METHOD dataProcessing : BOOL
VAR_INPUT
END_VAR
VAR
	i_CGResult:INT;
	i_HResult:INT;
	str1:STRING;
END_VAR
FOR logHandleArray_index:=1 TO logHandleArrayLength DO
	CASE nSocketType OF
	0://TCPIP server
		str1:=CONCAT(str1,BYTE_TO_HEXSTR(tcpipRecData.b1,2,FALSE));
		str1:=CONCAT(str1,' ');
		str1:=CONCAT(str1,BYTE_TO_HEXSTR(tcpipRecData.b2,2,FALSE));
		str1:=CONCAT(str1,' ');
		str1:=CONCAT(str1,BYTE_TO_HEXSTR(tcpipRecData.b3,2,FALSE));
		str1:=CONCAT(str1,' ');
		str1:=CONCAT(str1,BYTE_TO_HEXSTR(tcpipRecData.b4,2,FALSE));
		str1:=CONCAT(str1,' ');
		str1:=CONCAT(str1,BYTE_TO_HEXSTR(tcpipRecData.b5,2,FALSE));
		str1:=CONCAT(str1,' ');
		str1:=CONCAT(str1,BYTE_TO_HEXSTR(tcpipRecData.b6,2,FALSE));
		str1:=CONCAT(str1,' ');
		str1:=CONCAT(str1,BYTE_TO_HEXSTR(tcpipRecData.b7,2,FALSE));
		str1:=CONCAT(str1,' ');
		str1:=CONCAT(str1,BYTE_TO_HEXSTR(tcpipRecData.b8,2,FALSE));
		str1:=CONCAT(str1,' ');
		str1:=CONCAT(str1,BYTE_TO_HEXSTR(tcpipRecData.b9,2,FALSE));
		str1:=CONCAT(str1,' ');
		str1:=CONCAT(str1,BYTE_TO_HEXSTR(tcpipRecData.b10,2,FALSE));
		str1:=CONCAT(str1,' ');
		str1:=CONCAT(str1,BYTE_TO_HEXSTR(tcpipRecData.b11,2,FALSE));
		str1:=CONCAT(str1,' ');
		str1:=CONCAT(str1,BYTE_TO_HEXSTR(tcpipRecData.b12,2,FALSE));
		str1:=CONCAT(str1,' ');
		str1:=CONCAT(str1,BYTE_TO_HEXSTR(tcpipRecData.b13,2,FALSE));
		str1:=CONCAT(str1,' ');
		str1:=CONCAT(str1,BYTE_TO_HEXSTR(tcpipRecData.b14,2,FALSE));
		str1:=CONCAT(str1,' ');
		str1:=CONCAT(str1,BYTE_TO_HEXSTR(tcpipRecData.b15,2,FALSE));
		str1:=CONCAT(str1,' ');
		str1:=CONCAT(str1,BYTE_TO_HEXSTR(tcpipRecData.b16,2,FALSE));
		str1:=CONCAT(str1,' ');
		str1:=CONCAT(str1,BYTE_TO_HEXSTR(tcpipRecData.b17,2,FALSE));
		str1:=CONCAT(str1,' ');
		str1:=CONCAT(str1,BYTE_TO_HEXSTR(tcpipRecData.b18,2,FALSE));
		str1:=CONCAT(str1,' ');
		str1:=CONCAT(str1,BYTE_TO_HEXSTR(tcpipRecData.b19,2,FALSE));
		str1:=CONCAT(str1,' ');
		str1:=CONCAT(str1,BYTE_TO_HEXSTR(tcpipRecData.b20,2,FALSE));
//		logHandleArray[logHandleArray_index]^.append(CONCAT(CONCAT(CONCAT('Recevie From ', sTerminalName), ' -- '),str1));
	1://TCPIP client
		str1:=CONCAT(str1,BYTE_TO_HEXSTR(tcpipRecData.b1,2,FALSE));
		str1:=CONCAT(str1,' ');
		str1:=CONCAT(str1,BYTE_TO_HEXSTR(tcpipRecData.b2,2,FALSE));
		str1:=CONCAT(str1,' ');
		str1:=CONCAT(str1,BYTE_TO_HEXSTR(tcpipRecData.b3,2,FALSE));
		str1:=CONCAT(str1,' ');
		str1:=CONCAT(str1,BYTE_TO_HEXSTR(tcpipRecData.b4,2,FALSE));
		str1:=CONCAT(str1,' ');
		str1:=CONCAT(str1,BYTE_TO_HEXSTR(tcpipRecData.b5,2,FALSE));
		str1:=CONCAT(str1,' ');
		str1:=CONCAT(str1,BYTE_TO_HEXSTR(tcpipRecData.b6,2,FALSE));
		str1:=CONCAT(str1,' ');
		str1:=CONCAT(str1,BYTE_TO_HEXSTR(tcpipRecData.b7,2,FALSE));
		str1:=CONCAT(str1,' ');
		str1:=CONCAT(str1,BYTE_TO_HEXSTR(tcpipRecData.b8,2,FALSE));
		str1:=CONCAT(str1,' ');
		str1:=CONCAT(str1,BYTE_TO_HEXSTR(tcpipRecData.b9,2,FALSE));
		str1:=CONCAT(str1,' ');
		str1:=CONCAT(str1,BYTE_TO_HEXSTR(tcpipRecData.b10,2,FALSE));
		str1:=CONCAT(str1,' ');
		str1:=CONCAT(str1,BYTE_TO_HEXSTR(tcpipRecData.b11,2,FALSE));
		str1:=CONCAT(str1,' ');
		str1:=CONCAT(str1,BYTE_TO_HEXSTR(tcpipRecData.b12,2,FALSE));
		str1:=CONCAT(str1,' ');
		str1:=CONCAT(str1,BYTE_TO_HEXSTR(tcpipRecData.b13,2,FALSE));
		str1:=CONCAT(str1,' ');
		str1:=CONCAT(str1,BYTE_TO_HEXSTR(tcpipRecData.b14,2,FALSE));
		str1:=CONCAT(str1,' ');
		str1:=CONCAT(str1,BYTE_TO_HEXSTR(tcpipRecData.b15,2,FALSE));
		str1:=CONCAT(str1,' ');
		str1:=CONCAT(str1,BYTE_TO_HEXSTR(tcpipRecData.b16,2,FALSE));
		str1:=CONCAT(str1,' ');
		str1:=CONCAT(str1,BYTE_TO_HEXSTR(tcpipRecData.b17,2,FALSE));
		str1:=CONCAT(str1,' ');
		str1:=CONCAT(str1,BYTE_TO_HEXSTR(tcpipRecData.b18,2,FALSE));
		str1:=CONCAT(str1,' ');
		str1:=CONCAT(str1,BYTE_TO_HEXSTR(tcpipRecData.b19,2,FALSE));
		str1:=CONCAT(str1,' ');
		str1:=CONCAT(str1,BYTE_TO_HEXSTR(tcpipRecData.b20,2,FALSE));
//		logHandleArray[logHandleArray_index]^.append(CONCAT(CONCAT(CONCAT('Recevie From ', sTerminalName), ' -- '),str1));
	END_CASE
END_FOR

// 数据处理
readStateFlag:=TRUE;
volt:=TO_REAL((tcpipRecData.b10*256+tcpipRecData.b11)/4096.0)*10.0;
dworld:=tcpipRecData.b10*256+tcpipRecData.b11;
END_METHOD

ACTION Manual:
(*
rTrig_Version(CLK:=bTrig_Version);
IF rTrig_Version.Q THEN
	appendSend(0,0,E_CmdID_SW.SW_GetVer,0.0,0.0,0.0,0.0,0.0,0,'');
END_IF
*)
END_ACTION

METHOD PRIVATE popup : BOOL
VAR_INPUT
END_VAR
CASE popupStep OF
0:
	IF (sendPoint<endPoint OR passMax) AND bSendCondition THEN
		popupSendData:=sendDataArray[sendPoint];
		sendData(popupSendData);//此处是调用信息发送
		popupStep:=10;
		sendPoint:=sendPoint+1;
		IF sendPoint>(cNumEnd-1) THEN
			sendPoint:=1;
			passMax:=FALSE;
		END_IF
	END_IF
10:
	popupTON2(IN:=NOT popupTON2.Q, PT:=T#2S);
	IF NOT bSendCondition OR popupTON2.Q THEN
		popupTON2(IN:=FALSE);
		popupStep:=11;
	END_IF
11:
	IF bSendCondition THEN
		popupStep:=12;
	END_IF
	popupTON1(IN:=FALSE);
12:
	//popupTON1(IN:=NOT popupTON1.Q,PT:=T#10MS);
	popupTON1(IN:=NOT popupTON1.Q,PT:=TO_TIME(nQueueInterval));
	IF popupTON1.Q THEN
		popupStep:=0;
	END_IF
END_CASE
END_METHOD

METHOD ReadVoltage : BOOL
VAR_INPUT
END_VAR
appendSend(16#00,16#00,16#00,16#00,16#00,16#06,16#01,16#04,16#00,16#00,16#00,16#04,0,0,0,0,0,0,0,0,12);// 读进电压字符串
END_METHOD

METHOD PRIVATE sendData : BOOL
VAR_INPUT
	dataStruct	:struct_byte;
END_VAR
VAR
	str1:STRING;
END_VAR
IF bSendCondition AND bEnable THEN
	tcpipSendData.b1	:=dataStruct.b1;
	tcpipSendData.b2	:=dataStruct.b2;
	tcpipSendData.b3	:=dataStruct.b3;
	tcpipSendData.b4	:=dataStruct.b4;
	tcpipSendData.b5	:=dataStruct.b5;
	tcpipSendData.b6	:=dataStruct.b6;
	tcpipSendData.b7	:=dataStruct.b7;
	tcpipSendData.b8	:=dataStruct.b8;
	tcpipSendData.b9	:=dataStruct.b9;
	tcpipSendData.b10	:=dataStruct.b10;
	tcpipSendData.b11	:=dataStruct.b11;
	tcpipSendData.b12	:=dataStruct.b12;
	tcpipSendData.b13	:=dataStruct.b13;
	tcpipSendData.b14	:=dataStruct.b14;
	tcpipSendData.b15	:=dataStruct.b15;
	tcpipSendData.b16	:=dataStruct.b16;
	tcpipSendData.b17	:=dataStruct.b17;
	tcpipSendData.b18	:=dataStruct.b18;
	tcpipSendData.b19	:=dataStruct.b19;
	tcpipSendData.b20	:=dataStruct.b20;
	
	CASE nSocketType OF
	0://TCPIP server
		tcpipSendDataBuff_Server:=tcpipSendData;
		tcpipSendData:=tcpipSendDataClear;	
		tcpipServer.bSend:=TRUE;
	1://TCPIP client
		tcpipSendDataBuff_Client:=tcpipSendData;
		tcpipSendData:=tcpipSendDataClear;	
		tcpipClient.bSend:=TRUE;
	END_CASE
	
	FOR logHandleArray_index:=1 TO logHandleArrayLength DO
		CASE nSocketType OF
		0://TCPIP server
			str1:=CONCAT(str1,BYTE_TO_HEXSTR(tcpipSendDataBuff_Server.b1,2,FALSE));
			str1:=CONCAT(str1,' ');
			str1:=CONCAT(str1,BYTE_TO_HEXSTR(tcpipSendDataBuff_Server.b2,2,FALSE));
			str1:=CONCAT(str1,' ');
			str1:=CONCAT(str1,BYTE_TO_HEXSTR(tcpipSendDataBuff_Server.b3,2,FALSE));
			str1:=CONCAT(str1,' ');
			str1:=CONCAT(str1,BYTE_TO_HEXSTR(tcpipSendDataBuff_Server.b4,2,FALSE));
			str1:=CONCAT(str1,' ');
			str1:=CONCAT(str1,BYTE_TO_HEXSTR(tcpipSendDataBuff_Server.b5,2,FALSE));
			str1:=CONCAT(str1,' ');
			str1:=CONCAT(str1,BYTE_TO_HEXSTR(tcpipSendDataBuff_Server.b6,2,FALSE));
			str1:=CONCAT(str1,' ');
			str1:=CONCAT(str1,BYTE_TO_HEXSTR(tcpipSendDataBuff_Server.b7,2,FALSE));
			str1:=CONCAT(str1,' ');
			str1:=CONCAT(str1,BYTE_TO_HEXSTR(tcpipSendDataBuff_Server.b8,2,FALSE));
			str1:=CONCAT(str1,' ');
			str1:=CONCAT(str1,BYTE_TO_HEXSTR(tcpipSendDataBuff_Server.b9,2,FALSE));
			str1:=CONCAT(str1,' ');
			str1:=CONCAT(str1,BYTE_TO_HEXSTR(tcpipSendDataBuff_Server.b10,2,FALSE));
			str1:=CONCAT(str1,' ');
			str1:=CONCAT(str1,BYTE_TO_HEXSTR(tcpipSendDataBuff_Server.b11,2,FALSE));
			str1:=CONCAT(str1,' ');
			str1:=CONCAT(str1,BYTE_TO_HEXSTR(tcpipSendDataBuff_Server.b12,2,FALSE));
			str1:=CONCAT(str1,' ');
			str1:=CONCAT(str1,BYTE_TO_HEXSTR(tcpipSendDataBuff_Server.b13,2,FALSE));
			str1:=CONCAT(str1,' ');
			str1:=CONCAT(str1,BYTE_TO_HEXSTR(tcpipSendDataBuff_Server.b14,2,FALSE));
			str1:=CONCAT(str1,' ');
			str1:=CONCAT(str1,BYTE_TO_HEXSTR(tcpipSendDataBuff_Server.b15,2,FALSE));
			str1:=CONCAT(str1,' ');
			str1:=CONCAT(str1,BYTE_TO_HEXSTR(tcpipSendDataBuff_Server.b16,2,FALSE));
			str1:=CONCAT(str1,' ');
			str1:=CONCAT(str1,BYTE_TO_HEXSTR(tcpipSendDataBuff_Server.b17,2,FALSE));
			str1:=CONCAT(str1,' ');
			str1:=CONCAT(str1,BYTE_TO_HEXSTR(tcpipSendDataBuff_Server.b18,2,FALSE));
			str1:=CONCAT(str1,' ');
			str1:=CONCAT(str1,BYTE_TO_HEXSTR(tcpipSendDataBuff_Server.b19,2,FALSE));
			str1:=CONCAT(str1,' ');
			str1:=CONCAT(str1,BYTE_TO_HEXSTR(tcpipSendDataBuff_Server.b20,2,FALSE));
//			logHandleArray[logHandleArray_index]^.append(CONCAT(CONCAT(CONCAT('Send To ', sTerminalName), ' -- '),str1));
		1://TCPIP client
			str1:=CONCAT(str1,' ');
			str1:=CONCAT(str1,BYTE_TO_HEXSTR(tcpipSendDataBuff_Client.b1,2,FALSE));
			str1:=CONCAT(str1,' ');
			str1:=CONCAT(str1,BYTE_TO_HEXSTR(tcpipSendDataBuff_Client.b2,2,FALSE));
			str1:=CONCAT(str1,' ');
			str1:=CONCAT(str1,BYTE_TO_HEXSTR(tcpipSendDataBuff_Client.b3,2,FALSE));
			str1:=CONCAT(str1,' ');
			str1:=CONCAT(str1,BYTE_TO_HEXSTR(tcpipSendDataBuff_Client.b4,2,FALSE));
			str1:=CONCAT(str1,' ');
			str1:=CONCAT(str1,BYTE_TO_HEXSTR(tcpipSendDataBuff_Client.b5,2,FALSE));
			str1:=CONCAT(str1,' ');
			str1:=CONCAT(str1,BYTE_TO_HEXSTR(tcpipSendDataBuff_Client.b6,2,FALSE));
			str1:=CONCAT(str1,' ');
			str1:=CONCAT(str1,BYTE_TO_HEXSTR(tcpipSendDataBuff_Client.b7,2,FALSE));
			str1:=CONCAT(str1,' ');
			str1:=CONCAT(str1,BYTE_TO_HEXSTR(tcpipSendDataBuff_Client.b8,2,FALSE));
			str1:=CONCAT(str1,' ');
			str1:=CONCAT(str1,BYTE_TO_HEXSTR(tcpipSendDataBuff_Client.b9,2,FALSE));
			str1:=CONCAT(str1,' ');
			str1:=CONCAT(str1,BYTE_TO_HEXSTR(tcpipSendDataBuff_Client.b10,2,FALSE));
			str1:=CONCAT(str1,' ');
			str1:=CONCAT(str1,BYTE_TO_HEXSTR(tcpipSendDataBuff_Client.b11,2,FALSE));
			str1:=CONCAT(str1,' ');
			str1:=CONCAT(str1,BYTE_TO_HEXSTR(tcpipSendDataBuff_Client.b12,2,FALSE));
			str1:=CONCAT(str1,' ');
			str1:=CONCAT(str1,BYTE_TO_HEXSTR(tcpipSendDataBuff_Client.b13,2,FALSE));
			str1:=CONCAT(str1,' ');
			str1:=CONCAT(str1,BYTE_TO_HEXSTR(tcpipSendDataBuff_Client.b14,2,FALSE));
			str1:=CONCAT(str1,' ');
			str1:=CONCAT(str1,BYTE_TO_HEXSTR(tcpipSendDataBuff_Client.b15,2,FALSE));
			str1:=CONCAT(str1,' ');
			str1:=CONCAT(str1,BYTE_TO_HEXSTR(tcpipSendDataBuff_Client.b16,2,FALSE));
			str1:=CONCAT(str1,' ');
			str1:=CONCAT(str1,BYTE_TO_HEXSTR(tcpipSendDataBuff_Client.b17,2,FALSE));
			str1:=CONCAT(str1,' ');
			str1:=CONCAT(str1,BYTE_TO_HEXSTR(tcpipSendDataBuff_Client.b18,2,FALSE));
			str1:=CONCAT(str1,' ');
			str1:=CONCAT(str1,BYTE_TO_HEXSTR(tcpipSendDataBuff_Client.b19,2,FALSE));
			str1:=CONCAT(str1,' ');
			str1:=CONCAT(str1,BYTE_TO_HEXSTR(tcpipSendDataBuff_Client.b20,2,FALSE));
//			logHandleArray[logHandleArray_index]^.append(CONCAT(CONCAT(CONCAT('Send To ', sTerminalName), ' -- '),str1));
		END_CASE
	END_FOR
END_IF
END_METHOD

END_PROGRAM

// ---- POUs/Communication/PLC_String.TcPOU
PROGRAM PLC_String
VAR_INPUT
	nSocketType:UINT:=0;// socket 类型; 0 表示 server; 1 表示 client;
	sTerminalName:STRING;// 通讯对方名称 自定义
	sHost:STRING(20):='127.0.0.1';// 通讯IP地址; server时表示本地host; client时表示远程host
	nPort:UDINT:=8900;// 通讯端口号;
	bEnable:BOOL:=TRUE;// 通讯启用\禁用连接
	sSendSuffix:STRING:='';//此处可统一添加发送后缀字符 $R$N
	nQueueInterval:UDINT:=50;// 发送队列时间间隔 单位ms
	logHandleArray:ARRAY [1..5] OF POINTER TO printLogModule_EX;// log 操作 handle 数组
	logHandleArrayLength:UINT:=0;// log 操作 handle 数组长度, 不超过5
END_VAR
VAR_OUTPUT
	bSendCondition	:BOOL;//可发送条件
	bSocketConnected:BOOL;//连接状态
END_VAR
VAR CONSTANT
	cNumBegin		:DINT:=1;
	cNumEnd			:DINT:=100;
END_VAR
VAR
	sendDataArray	:ARRAY [cNumBegin..cNumEnd] OF STRING(255);
	length			:DINT:=0;
	endPoint		:DINT:=cNumBegin;
	popupSendData	:STRING(255);
	//popup
	popupStep		:UINT:=0;
	popupTON1		:TON;
	popupTON2		:TON;
	iPopup			:DINT:=0;
	_PopupLength	:DINT:=0;
END_VAR
VAR
	tcpipClient					:tcpipClientModule_EX;
	tcpipServer					:tcpipServerModule_EX;////定义服务器对象
	
	tcpipSendDataBuff_Server	:STRING(255);//发送数据 Buff server
	tcpipSendDataBuff_Client	:STRING(255);//发送数据 Buff client
	
	tcpipSendDataClear			:STRING(255);//发送数据 清空
	tcpipSendData				:STRING(255);//发送数据
	
	tcpipRecDataBuff_Server		:STRING(255);//已接收数据 Buff server
	tcpipRecDataBuff_Client		:STRING(255);//已接收数据 Buff client
	
	tcpipRecDataClear			:STRING(255);//已接收数据 清空
	tcpipRecData				:STRING(255);//已接收数据
	
	tcpConnectR_Trig			:R_Trig;//初始连接上升沿
	tcpConnectF_Trig			:F_Trig;//初始连接下降沿
	registerStep				:UDINT;//ALC注册控制步
	registerTON					:TON;//ALC注册延时
	
	logHandleArray_index		:UINT:=1;
END_VAR
VAR
	bTrig_Start:BOOL;
	rTrig_Start:R_TRIG;
	tTrig_Start:TON;
	
	bTrig_Stop:BOOL;
	rTrig_Stop:R_TRIG;
	tTrig_Stop:TON;
	
	bTrig_Reset:BOOL;
	rTrig_Reset:R_TRIG;
	tTrig_Reset:TON;
	
	
	bTrig_Init:BOOL;
	rTrig_Init:R_TRIG;
	
	bTrig_All_Home:BOOL;
	rTrig_All_Home:R_TRIG;
	
	bTrig_Z_Safe:BOOL;
	rTrig_Z_Safe:R_TRIG;
	
	bTrig_P_Pos_:BOOL;
	rTrig_P_Pos_:R_TRIG;
	nTrig_P_Pos_TrayNum:UINT:=1;
	nTrig_P_Pos_RowNum:UINT:=1;
	
	bTrig_Move_P_:BOOL;
	rTrig_Move_P_:R_TRIG;
	nTrig_Move_P_TrayNum:UINT:=1;
	nTrig_Move_P_RowNum:UINT:=1;
	nTrig_Move_P_PosNum:UINT:=1;
	findposstart	:INT;
	findposend		:INT;
	find_pos		:INT;
	recStrTemp		:STRING(255);
END_VAR


CASE nSocketType OF
0://TCPIP server
	tcpipServer(
		sSrvNetId:= , 
		sLocalHost:=sHost , 
		nLocalPort:=nPort , 
		bStartConnect:=bEnable , 
		tcpipSDataLen:=TO_UDINT(LEN(tcpipSendDataBuff_Server)) , 
		tcpipSData:=ADR(tcpipSendDataBuff_Server) , 
		bSend:= , 
		tcpipRecDataLen:=SIZEOF(tcpipRecDataBuff_Server) , 
		tcpipRecData:=ADR(tcpipRecDataBuff_Server) , 
		bAccepted=> , 
		bSendBusy=> , 
		bRecData=> );
	bSendCondition:=tcpipServer.bAccepted AND NOT tcpipServer.bSendBusy;
	//TCPIP连接
	bSocketConnected:=tcpipServer.bAccepted;
	IF NOT tcpipServer.bAccepted THEN
		length:=0;
		endPoint:=cNumBegin;
	END_IF
	tcpConnectR_Trig(CLK:=tcpipServer.bAccepted);
	tcpConnectF_Trig(CLK:=tcpipServer.bAccepted);

1://TCPIP client
	tcpipClient(
		sSrvNetId:= , 
		sRemoteHost:=sHost , 
		nRemotePort:=nPort , 
		bStartConnect:=bEnable , 
		tcpipSDataLen:=TO_UDINT(LEN(tcpipSendDataBuff_Client)) , 
		tcpipSData:=ADR(tcpipSendDataBuff_Client) , 
		bSend:= , 
		tcpipRecDataLen:=SIZEOF(tcpipRecDataBuff_Client) , 
		tcpipRecData:=ADR(tcpipRecDataBuff_Client) , 
		bConnected=> , 
		bSendBusy=> , 
		bRecData=> );
	bSendCondition:=tcpipClient.bConnected AND NOT tcpipClient.bSendBusy;
	//TCPIP连接
	bSocketConnected:=tcpipClient.bConnected;
	IF NOT tcpipClient.bConnected THEN
		length:=0;
		endPoint:=cNumBegin;
	END_IF
	tcpConnectR_Trig(CLK:=tcpipClient.bConnected);
	tcpConnectF_Trig(CLK:=tcpipClient.bConnected);
END_CASE

IF tcpConnectR_Trig.Q THEN
	FOR logHandleArray_index:=1 TO logHandleArrayLength DO
		logHandleArray[logHandleArray_index]^.append(CONCAT(sTerminalName, ' has been connected'));
	END_FOR
	registerStep:=10;
END_IF
IF tcpConnectF_Trig.Q THEN
	FOR logHandleArray_index:=1 TO logHandleArrayLength DO
		logHandleArray[logHandleArray_index]^.append(CONCAT(sTerminalName, ' has been disconnected'));
	END_FOR
	registerStep:=0;
END_IF
//数据接收处理
CASE nSocketType OF
0://TCPIP server
	IF tcpipServer.bRecData THEN
		tcpipRecData:=tcpipRecDataBuff_Server;//buff转存
		tcpipRecDataBuff_Server:=tcpipRecDataClear;//转存之后清空buff
		dataProcessing();
	END_IF
1://TCPIP client
	IF tcpipClient.bRecData THEN
		tcpipRecData:=tcpipRecDataBuff_Client;//buff转存
		tcpipRecDataBuff_Client:=tcpipRecDataClear;//转存之后清空buff
		dataProcessing();
	END_IF
END_CASE


popup();

CASE registerStep OF
0:
	//Ready
END_CASE

ACTION ACT_dataProcessing_DOE:
//(*LoadCCD3*)
//	recStrFilArrSocket[1]:='CoaxialCCD1:';
//	recStrFilArrSocket[2]:='DUTTopX:';
//	recStrFilArrSocket[3]:='DUTTopY:';
//	recStrFilArrSocket[4]:='DUTBottomX:';
//	recStrFilArrSocket[5]:='DUTBottomY:';
//	recStrFilArrSocket[6]:='SocketTopX:';
//	recStrFilArrSocket[7]:='SocketTopY:';
//	recStrFilArrSocket[8]:='SocketBottomX:';
//	recStrFilArrSocket[9]:='SocketBottomY:';
//	recStrFilArrSocket[10]:='ModelAngle:';
	
//	recStrTemp:='';
//	find_pos:=FIND(tcpipRecData, recStrFilArrSocket[1]);
//	IF find_pos>0 THEN
//		findposstart:=find_pos;
//		find_pos:=0;
//		find_pos:=FIND(tcpipRecData, ';');
//		IF find_pos>0 THEN
//			findposend:=find_pos;
//			find_pos:=0;
//		END_IF
//		recPosArrSocket_G_CCD1[1]:=STRING_TO_LREAL(MID(tcpipRecData,findposend-findposstart-(len(recStrFilArrSocket[1])+len(recStrFilArrSocket[2])),findposstart+len(recStrFilArrSocket[1])+len(recStrFilArrSocket[2])));
//		recStrTemp:=DELETE(tcpipRecData,findposend-findposstart+1,findposstart);
//		find_pos:=0;
//		findposstart:=1;
//		find_pos:=FIND(recStrTemp, ';');
//		IF find_pos>0 THEN
//			findposend:=find_pos;
//			find_pos:=0;
//		END_IF
//		recPosArrSocket_G_CCD1[2]:=STRING_TO_LREAL(MID(recStrTemp,findposend-findposstart-len(recStrFilArrSocket[3]),findposstart+len(recStrFilArrSocket[3])));
//		recStrTemp:=DELETE(recStrTemp,findposend-findposstart+1,findposstart);
//		find_pos:=0;
//		findposstart:=1;
//		find_pos:=FIND(recStrTemp, ';');
//		IF find_pos>0 THEN
//			findposend:=find_pos;
//			find_pos:=0;
//		END_IF
//		recPosArrSocket_G_CCD1[3]:=STRING_TO_LREAL(MID(recStrTemp,findposend-findposstart-len(recStrFilArrSocket[4]),findposstart+len(recStrFilArrSocket[4])));
//		recStrTemp:=DELETE(recStrTemp,findposend-findposstart+1,findposstart);
//		find_pos:=0;
//		findposstart:=1;
//		find_pos:=FIND(recStrTemp, ';');
//		IF find_pos>0 THEN
//			findposend:=find_pos;
//			find_pos:=0;
//		END_IF
//		recPosArrSocket_G_CCD1[4]:=STRING_TO_LREAL(MID(recStrTemp,findposend-findposstart-len(recStrFilArrSocket[5]),findposstart+len(recStrFilArrSocket[5])));
//		recStrTemp:=DELETE(recStrTemp,findposend-findposstart+1,findposstart);
//		find_pos:=0;
//		findposstart:=1;
//		find_pos:=FIND(recStrTemp, ';');
//		IF find_pos>0 THEN
//			findposend:=find_pos;
//			find_pos:=0;
//		END_IF
//		recPosArrSocket_G_CCD1[5]:=STRING_TO_LREAL(MID(recStrTemp,findposend-findposstart-len(recStrFilArrSocket[6]),findposstart+len(recStrFilArrSocket[6])));
//		recStrTemp:=DELETE(recStrTemp,findposend-findposstart+1,findposstart);
//		find_pos:=0;
//		findposstart:=1;
//		find_pos:=FIND(recStrTemp, ';');
//		IF find_pos>0 THEN
//			findposend:=find_pos;
//			find_pos:=0;
//		END_IF
//		recPosArrSocket_G_CCD1[6]:=STRING_TO_LREAL(MID(recStrTemp,findposend-findposstart-len(recStrFilArrSocket[7]),findposstart+len(recStrFilArrSocket[7])));
//		recStrTemp:=DELETE(recStrTemp,findposend-findposstart+1,findposstart);
//		find_pos:=0;
//		findposstart:=1;
//		find_pos:=FIND(recStrTemp, ';');
//		IF find_pos>0 THEN
//			findposend:=find_pos;
//			find_pos:=0;
//		END_IF
//		recPosArrSocket_G_CCD1[7]:=STRING_TO_LREAL(MID(recStrTemp,findposend-findposstart-len(recStrFilArrSocket[8]),findposstart+len(recStrFilArrSocket[8])));
//		recStrTemp:=DELETE(recStrTemp,findposend-findposstart+1,findposstart);
//		find_pos:=0;
//		findposstart:=1;
//		find_pos:=FIND(recStrTemp, ';');
//		IF find_pos>0 THEN
//			findposend:=find_pos;
//			find_pos:=0;
//		END_IF
//		recPosArrSocket_G_CCD1[8]:=STRING_TO_LREAL(MID(recStrTemp,findposend-findposstart-len(recStrFilArrSocket[9]),findposstart+len(recStrFilArrSocket[9])));
//		recStrTemp:=DELETE(recStrTemp,findposend-findposstart+1,findposstart);
//		find_pos:=0;
//		findposstart:=1;
//		find_pos:=FIND(recStrTemp, ';');
//		IF find_pos>0 THEN
//			findposend:=find_pos;
//			find_pos:=0;
//		END_IF
//		recPosArrSocket_G_CCD1[9]:=STRING_TO_LREAL(MID(recStrTemp,findposend-findposstart-len(recStrFilArrSocket[10]),findposstart+len(recStrFilArrSocket[10])));
//		recStrTemp:=DELETE(recStrTemp,findposend-findposstart+1,findposstart);
//		recCCDResultArr[3]:=TRUE;
//	END_IF
END_ACTION

METHOD appendSend : BOOL
VAR_INPUT
	str			:STRING(255);
END_VAR
VAR
	suffix					:STRING;
	strTemp_appendSend		:STRING(255);
END_VAR

IF endPoint>(cNumEnd-1) THEN
	RETURN;
END_IF
suffix:=sSendSuffix;//此处可统一添加发送后缀字符 $R$N

strTemp_appendSend:=CONCAT(str,suffix);
sendDataArray[endPoint]:=strTemp_appendSend;

endPoint:=endPoint+1;
length:=endPoint-cNumBegin;
END_METHOD

METHOD dataProcessing : BOOL
VAR_INPUT
END_VAR
VAR
END_VAR
FOR logHandleArray_index:=1 TO logHandleArrayLength DO
	CASE nSocketType OF
	0://TCPIP server
		logHandleArray[logHandleArray_index]^.append(CONCAT(CONCAT(CONCAT('Recevie From ', sTerminalName), ' -- '),tcpipRecData));
	1://TCPIP client
		logHandleArray[logHandleArray_index]^.append(CONCAT(CONCAT(CONCAT('Recevie From ', sTerminalName), ' -- '),tcpipRecData));
	END_CASE
END_FOR
findposend:=0;
find_pos:=0;
ACT_dataProcessing_DOE();
END_METHOD

METHOD PRIVATE popup : BOOL
VAR_INPUT
END_VAR
CASE popupStep OF
0:
	IF length>0 AND bSendCondition THEN
		_PopupLength:=length;
		popupSendData:=sendDataArray[cNumBegin];
		FOR iPopup:=cNumBegin TO (_PopupLength-1) DO
			sendDataArray[iPopup]:=sendDataArray[iPopup+1];
		END_FOR
		endPoint:=endPoint-1;
		length:=endPoint-cNumBegin;
		sendData(popupSendData);//此处是调用信息发送
		popupStep:=10;
	END_IF
10:
	popupTON2(IN:=NOT popupTON2.Q, PT:=T#2S);
	IF NOT bSendCondition OR popupTON2.Q THEN
		popupTON2(IN:=FALSE);
		popupStep:=11;
	END_IF
11:
	IF bSendCondition THEN
		popupStep:=12;
	END_IF
	popupTON1(IN:=FALSE);
12:
	//popupTON1(IN:=NOT popupTON1.Q,PT:=T#10MS);
	popupTON1(IN:=NOT popupTON1.Q,PT:=TO_TIME(nQueueInterval));
	IF popupTON1.Q THEN
		popupStep:=0;
	END_IF
END_CASE
END_METHOD

METHOD PRIVATE sendData : BOOL
VAR_INPUT
	dataStruct	:STRING(255);
END_VAR
IF bSendCondition AND bEnable THEN
	tcpipSendData:=dataStruct;
	
	CASE nSocketType OF
	0://TCPIP server
		tcpipSendDataBuff_Server:=tcpipSendData;
		tcpipSendData:=tcpipSendDataClear;	
		tcpipServer.bSend:=TRUE;
	1://TCPIP client
		tcpipSendDataBuff_Client:=tcpipSendData;
		tcpipSendData:=tcpipSendDataClear;	
		tcpipClient.bSend:=TRUE;
	END_CASE
	
	FOR logHandleArray_index:=1 TO logHandleArrayLength DO
		CASE nSocketType OF
		0://TCPIP server
			logHandleArray[logHandleArray_index]^.append(CONCAT(CONCAT(CONCAT('Send To ', sTerminalName), ' -- '),tcpipSendDataBuff_Server));
		1://TCPIP client
			logHandleArray[logHandleArray_index]^.append(CONCAT(CONCAT(CONCAT('Send To ', sTerminalName), ' -- '),tcpipSendDataBuff_Client));
		END_CASE
	END_FOR
END_IF
END_METHOD

END_PROGRAM

// ---- POUs/Other/MachineState/MachineStatePOU.TcPOU
PROGRAM MachineStatePOU
VAR
	
	itemp: INT;
	forceStop:BOOL;
	forceStopTON:TON;
END_VAR
VAR
	//fbMachineState		:FB_MachineState;
	//
	start_R_Trig						:R_Trig;
	start_TON							:TON;
	start_R_Trig1						:R_Trig;
	//
	stop_F_Trig							:F_Trig;
	stop_TON							:TON;
	//
	reset_TON							:TON;
	reset_TimeoutTON					:TON;
	reset_R_Trig						:R_Trig;
	reset_F_Trig						:F_Trig;
	//
	e_stop_F_Trig						:F_Trig;
	e_stop_TON							:TON;
	//
	ErrorAbort_TON						:TON;
	
	//error
	ErrorR_Trig							:R_Trig;
	ErrorF_Trig							:F_Trig;
	ton1:TON;
	t1:TON;
END_VAR

fbMachineState(
	RunningState:= gRunningState, 
	HMI_E_Stop:= , 
	HMI_Start:= , 
	HMI_Stop:= , 
	HMI_Reset:= , 
	HMI_EnableBuzzer:= , 
	HMI_AllStop:= , 
	HMI_Version:= gVersion, 
	Actual_E_Stop:= gMachineUtility.I_EStop, 
	Actual_Start:= gMachineUtility.I_Start, 
	Actual_Stop:= gMachineUtility.I_Stop, 
	Actual_Reset:= gMachineUtility.I_Reset, 
	iLanguage:= TO_UINT(gCNErrShow),
	E_Stop=> , 
	Reset=> , 
	Stop=> , 
	Start=> , 
	StartLamp=> gMachineUtility.O_StartLamp, 
	StopLamp=> gMachineUtility.O_StopLamp, 
	ResetLamp=> gMachineUtility.O_ResetLamp, 
	RedLamp=> gMachineUtility.O_RedLamp, 
	GreenLamp=> gMachineUtility.O_GreenLamp, 
	YellowLamp=> gMachineUtility.O_YellowLamp, 
	Buzzer=> gMachineUtility.O_Buzzer, 
	AllStop=> , 
	RunStateTxt=> );
IF fbMachineState.AllStop AND MAIN.tInit.Q THEN
	gErrorAbort:=TRUE;
	MainRunPOU.allAxisStop();
END_IF
//////////////////////////////////////////////////////////////////////////////
(* Start *)
	IF start_R_Trig.Q THEN//短按上升沿从暂停恢复自动 或者 切换控制模式为eAutoCtrMode
		IF (RunningStatus.ePauseState=gRunningState) AND (gAutoRunningFlag)
			AND ControlMode.eAutoCtrMode=gCtrlMode THEN
			gRunningState:=RunningStatus.eAutoState;//进入自动运行状态
		END_IF
		IF ControlMode.eAutoCtrMode<>gCtrlMode AND NOT gAutoRunningFlag AND NOT(RunningStatus.eHomeState=gRunningState) THEN
//			gCtrlMode:=ControlMode.eAutoCtrMode;
		END_IF
	END_IF
	start_R_Trig(CLK:=fbMachineState.Start);
	
	IF start_R_Trig1.Q THEN//长按3s上升沿进入自动
		IF (RunningStatus.eManualState=gRunningState) AND NOT gAutoRunningFlag
			AND ControlMode.eManualCtrMode=gCtrlMode THEN
			gRunningState:=RunningStatus.eAutoState;//进入自动运行状态
			gAutoRunningFlag:=TRUE;
		ELSE
			;
		END_IF
	END_IF
	start_TON(IN:=fbMachineState.Start, PT:=T#3000MS);
	start_R_Trig1(CLK:=start_TON.Q);
(* Stop *)
	IF stop_F_Trig.Q THEN//短按下降沿进入暂停
		IF (RunningStatus.eAutoState=gRunningState) AND (gAutoRunningFlag)
			AND ControlMode.eAutoCtrMode=gCtrlMode THEN
			gRunningState:=RunningStatus.ePauseState;//进入暂停状态
		END_IF
	END_IF
	forceStopTON(IN:=forceStop AND NOT forceStopTON.Q , PT:=T#2S , Q=> , ET=> );//强制停止报错
	IF forceStopTON.Q THEN
		;;
	END_IF
	stop_F_Trig(CLK:=fbMachineState.Stop);
	
	stop_TON(IN:=fbMachineState.Stop, PT:=T#3000MS);//自动运行中长按stop按钮退出自动
	IF stop_TON.Q THEN//长按3s退出自动
		IF (gAutoRunningFlag) AND ControlMode.eAutoCtrMode=gCtrlMode THEN
			gAutoRunningFlag:=FALSE;
		END_IF
		IF NOT gAutoRunningFlag AND ControlMode.eManualCtrMode<>gCtrlMode THEN
			gCtrlMode:=ControlMode.eManualCtrMode;
			IF RunningStatus.eErrorState<>gRunningState THEN
				gRunningState:=RunningStatus.eManualState;
			END_IF
		END_IF
		//加入回原点长按停止,复原状态
		IF NOT gAutoRunningFlag AND (gRunningState=RunningStatus.eHomeState) THEN
			gCtrlMode:=ControlMode.eManualCtrMode;
			gRunningState:=RunningStatus.eManualState;
			
		END_IF
	END_IF
(* reset *)
	reset_R_Trig(CLK:=fbMachineState.Reset);
	reset_F_Trig(CLK:=fbMachineState.Reset);
	IF reset_R_Trig.Q  THEN//短按上升沿清除错误
		errorMonitor.resetFunc();//报错清除
		IF (*ControlMode.eAutoCtrMode<>gCtrlMode AND*) NOT gAutoRunningFlag AND (gRunningState<>RunningStatus.eHomeState) THEN
			gRunningState:=RunningStatus.eManualState;//进入手动运行状态
		ELSE
			;
			//gRunningState:=RunningStatus.ePauseState;//进入暂停状态
		END_IF		
	END_IF
	IF reset_R_Trig.Q AND RunningStatus.eErrorState=gRunningState THEN//短按上升沿清除错误--主要在自动模式下起作用
		errorMonitor.resetFunc();//报错清除
		gRunningState:=RunningStatus.ePauseState;//进入暂停状态
	END_IF
	//与复位按钮无关
	IF (RunningStatus.eHomeState=gRunningState) (*OR Home_POU.busy*)  THEN//等待回原点完成
		reset_TimeoutTON(IN:=NOT reset_TimeoutTON.Q,PT:=T#300S);
		IF reset_TimeoutTON.Q THEN
			error_Trigger(2);//回原点超时
			gRunningState:=RunningStatus.eManualState;
		END_IF
//		IF Home_POU.done AND NOT gAutoRunningFlag THEN//回原完成时，是否需要回到手动状态？
//			gRunningState:=RunningStatus.eManualState;
//		END_IF
//		IF Home_POU.errDone AND NOT gAutoRunningFlag THEN
//			error_Trigger(3);//回原点错误
//		END_IF
	ELSE
		reset_TimeoutTON(IN:=FALSE);
	END_IF
	IF reset_TON.Q AND reset_F_Trig.Q (*AND NOT Home_POU.busy *)THEN//长按下降沿整机回零
		IF ControlMode.eManualCtrMode=gCtrlMode AND (RunningStatus.eManualState=gRunningState) THEN	
			gRunningState:=RunningStatus.eHomeState;
//			Home_POU.Act_init_status();//触发整机回零处理
//			Home_POU.Act_Ex();
		END_IF
	END_IF
	reset_TON(IN:=fbMachineState.Reset, PT:=T#3S);
(* E-stop *)
	e_stop_F_Trig(CLK:=fbMachineState.E_Stop);
	IF e_stop_F_Trig.Q AND MAIN.tInit.Q THEN//下降沿报错
		gAutoRunningFlag:=FALSE;
		gCtrlMode:=ControlMode.eManualCtrMode;
		gErrorAbort:=TRUE;
		error_Trigger(1);//急停报警
		gLog.append_EX(" 急停按下");
	END_IF
	IF NOT fbMachineState.E_Stop THEN
		gRunningState:=RunningStatus.eErrorState;//进入Error状态
	END_IF
	e_stop_TON(IN:=NOT fbMachineState.E_Stop AND NOT fbMachineState.Reset, PT:=T#500MS);
	IF e_stop_TON.Q AND MAIN.tInit.Q THEN
		gAutoRunningFlag:=FALSE;
		gErrorAbort:=TRUE;
		e_stop_TON(IN:=FALSE);
		//gErrTxtShow:=errorMonitor.getErrTXT(1);//急停报警显示
		//gErrWTxtShow:=errorMonitor.getErrWTXT(1);//急停报警显示
		MainRunPOU.allAxisStop();
	END_IF
(* Abort *)
	ErrorAbort_TON(IN:=gErrorAbort,PT:=T#5000MS);
	IF ErrorAbort_TON.Q THEN
		gErrorAbort:=FALSE;
		ErrorAbort_TON(IN:=FALSE);
	END_IF
//////////////////////////////////////////////////////////////////////////////
IF gAutoRunningFlag THEN
	gCtrlMode:=ControlMode.eAutoCtrMode;
END_IF
//////////////////////////////////////////////////////////////////////////////
t1(IN:=(NOT gAutoRunningFlag OR gCtrlMode<>ControlMode.eManualCtrMode) AND
	(gICP.LoadLockGauge.error OR
	 gICP.ChamberGauge.error OR
	 gICP.AIMGauge.error OR
	 gICP.TBGauge.error OR
	 gICP.ForeLineGauge.error OR
	gICP.ChamberGauge.outputValue1>700.0 OR
	gICP.TBGauge.outputValue>500.0 OR
	(gICP.ForeLineGauge.outputValue>500.0 AND NOT gICP.FastPummingExtRelay AND NOT gICP.SlowPummingExtRelay)),PT:=T#2S);
IF t1.Q THEN
	gRoughRemain:=FALSE;// 粗抽记忆
END_IF


//ErrorR_Trig(CLK:=(gRunningState=RunningStatus.eErrorState) AND gAutoRunningFlag , Q=> );
//ErrorF_Trig(CLK:=(gRunningState=RunningStatus.eErrorState) AND gAutoRunningFlag, Q=> );

//ErrorR_Trig(CLK:=(gRunningState=RunningStatus.eErrorState) AND gCtrlMode=2, Q=> );//自动的时候报错
//ErrorF_Trig(CLK:=(gRunningState=RunningStatus.eErrorState) AND gCtrlMode=2, Q=> );//自动恢复报错

//IF ErrorR_Trig.Q THEN//报错停止操作
//	AllPause:=TRUE;
//END_IF
//IF ErrorF_Trig.Q THEN
//	;
//END_IF

END_PROGRAM

// ---- POUs/MAIN.TcPOU
PROGRAM MAIN
VAR_INPUT
	tInit:TON;
END_VAR
VAR
	DelayStartGetSystemTime:TON;
	DelayFlagGetSystemTime:BOOL:=TRUE;
	fbGetLocalAmsNetId:FB_GetLocalAmsNetId;
	r1:r_trig;
	elm:STRING;
END_VAR

tInit(IN:= TRUE, PT:= T#5S, Q=> , ET=> );
GetSystemTime();// 获取系统时钟
ups_CX51X0();//UPS掉电保存
MainParComfer_HMI();//CPH-主界面参数传递
MainRunPOU();//实例化、函数调用等内容
CloseAllSocket();//关闭所有Socket接口
ServicesRefreshPOU();//服务重启
r1(CLK:=gAutoRunningFlag AND (gRunningState=RunningStatus.eErrorState));
IF r1.Q THEN
	gDownTimeLog.append_EX(WCONCAT("Step,Current error,",gErrWTxtShow));//仅打印到DownTime信息中，方便查询错误信息
END_IF

//PageChange();
gCurrentUser:=VisuUserManagement.g_VisuLoginProviderManager.m_arrLoginProvider[0].stUserName;
//VisuUserManagement.g_VisuLoginProviderManager.m_arrLoginProvider[1].stUserName;
//VisuUserManagement.g_VisuLoginProviderManager.m_arrLoginProvider[2].stUserName;
//VisuUserManagement.g_VisuLoginProviderManager.m_arrLoginProvider[3].stUserName;

METHOD changePage : BOOL
VAR_INPUT
	page:INT;
END_VAR
VAR
	itemp:INT;
END_VAR
//FOR itemp:=1 TO SIZEOF(gWindowsPageBt) DO
//	IF itemp<>page THEN
//		gWindowsPageBt[itemp]:=FALSE;
//	ELSE
//		gWindowsPageBt[itemp]:=TRUE;
//	END_IF
//END_FOR
END_METHOD

ACTION GetSystemNetId:
////获取系统ID先启动
//DelayStartGetSystemTime(IN:=DelayFlagGetSystemTime , PT:=T#0.5S , Q=> , ET=> );
//IF DelayStartGetSystemTime.Q THEN
//	DelayFlagGetSystemTime:=FALSE;
//	fbGetLocalAmsNetId(
//		 bExecute:=TRUE, 
//		 tTimeOut:= , 
//		 bBusy=> , 
//		 bError=> , 
//		 nErrId=> , 
//		 AddrString=> , 
//		 AddrBytes=> );
//END_IF
//IF DelayFlagGetSystemTime THEN
//	RETURN;
//END_IF
//fbGetLocalAmsNetId(
//	 bExecute:=FALSE, 
//	 tTimeOut:= , 
//	 bBusy=> , 
//	 bError=> , 
//	 nErrId=> , 
//	 AddrString=> , 
//	 AddrBytes=> );
//g_sAmsNetId:=fbGetLocalAmsNetId.AddrString;
END_ACTION

ACTION GetSystemTime:
// 获取系统NetID;有时间延时启动的效果
// 获取系统ID先启动
DelayStartGetSystemTime(IN:=DelayFlagGetSystemTime , PT:=T#0.5S , Q=> , ET=> );
IF DelayStartGetSystemTime.Q THEN
	DelayFlagGetSystemTime:=FALSE;
	fbGetLocalAmsNetId(
		 bExecute:=TRUE, 
		 tTimeOut:= , 
		 bBusy=> , 
		 bError=> , 
		 nErrId=> , 
		 AddrString=> , 
		 AddrBytes=> );
END_IF
IF DelayFlagGetSystemTime THEN
	RETURN;
END_IF
fbGetLocalAmsNetId(
	 bExecute:=FALSE, 
	 tTimeOut:= , 
	 bBusy=> , 
	 bError=> , 
	 nErrId=> , 
	 AddrString=> , 
	 AddrBytes=> );
g_sAmsNetId:=fbGetLocalAmsNetId.AddrString;
END_ACTION

ACTION PageChange:
//elm:=VisuElemsWinControls.CURRENTVISU;
//IF (elm='Main' OR elm='Auto_Main') THEN
//	MAIN.changePage(1);
//END_IF

//IF (elm='Recipe_Main') THEN
//	MAIN.changePage(2);
//END_IF

//IF (elm='IO_Main') THEN
//	MAIN.changePage(3);
//END_IF

//IF (elm='Log_Main') THEN
//	MAIN.changePage(4);
//END_IF

//IF (elm='Config_Main') THEN
//	MAIN.changePage(5);
//END_IF

//IF (elm='Loadding_Main') THEN
//	MAIN.changePage(6);
//END_IF
END_ACTION

END_PROGRAM

// ---- POUs/Other/MachineState/MainParComfer_HMI.TcPOU
PROGRAM MainParComfer_HMI
VAR
END_VAR

MainFramDUT.ComName:='GIDEON';//公司名称;
MainFramDUT.ProjectName:='ICP_01';//项目名称	
MainFramDUT.ShowTime:=g_SystemTime;//当前时间显示变量
//按钮灯
MainFramDUT.StartLamp:=fbMachineState.StartLamp;//启面急停动指示
MainFramDUT.ResetLamp:=fbMachineState.ResetLamp;//复面急停位指示
MainFramDUT.StopLamp:=fbMachineState.StopLamp;//停面急停止，报错指示
	
fbMachineState.HMI_E_Stop:=MainFramDUT.E_Stop;//界面急停显示
fbMachineState.HMI_Start:=MainFramDUT.Start;//界面启动
fbMachineState.HMI_Reset:=MainFramDUT.Reset;//界面复位
fbMachineState.HMI_Stop:=MainFramDUT.Stop;//界面停止
//三色灯
MainFramDUT.GreenLamp:=fbMachineState.GreenLamp;//绿灯
MainFramDUT.RedLamp:=fbMachineState.RedLamp;//红灯
MainFramDUT.YellowLamp:=fbMachineState.YellowLamp;//黄灯
//MainFramDUT.Loading:=;//界面登录
//MainFramDUT.Quit:=;//界面退出
MainFramDUT.versions:=gVersion;//版本号传递
MainFramDUT.RunStateTxt:=fbMachineState.RunStateTxtS;//版本号传递
MainFramDUT.ErrWTxtShow:=gErrWTxtShow;//版本号传递

END_PROGRAM

// ---- POUs/BaseModule/TcpIpModule_EX/CloseAllSocket.TcPOU
//在PLC 重新启动的时候 关闭所以Socket
PROGRAM CloseAllSocket
VAR
	fbSocketCloseAll : FB_SocketCloseAll;
    bCloseAll        : BOOL := TRUE;
	tInit 			 : TON;
END_VAR

tInit(IN:=TRUE , PT:=T#10MS , Q=> , ET=> );
IF NOT tInit.Q THEN
	fbSocketCloseAll( bExecute:= FALSE );
	RETURN;
END_IF

IF bCloseAll THEN(*On PLC reset or program download close all old connections *)
    bCloseAll := FALSE;
	fbSocketCloseAll(
		sSrvNetId:= '', 
		bExecute:= TRUE, 
		tTimeout:= T#10S, 
		bBusy=> , 
		bError=> , 
		nErrId=> );
ELSE
    fbSocketCloseAll( bExecute:= FALSE );
END_IF

ACTION VersionLog:
(*
版本: V1.0.0.0
说明:
	1. 首个版本
//**************************************************//
版本: V1.0.0.1
说明:
	1. 上电后延时关闭所有旧的连接
//**************************************************//
*)
END_ACTION

END_PROGRAM

// ---- POUs/Communication/ServicesRefreshPOU.TcPOU
PROGRAM ServicesRefreshPOU
VAR_OUTPUT
	bDone:BOOL;
	bErrDone:BOOL;
	sErrTxt:STRING;
END_VAR
VAR
	bInit:BOOL;
	tInit:TON;
	nStep:INT;
	fbNT_StartProcess:NT_StartProcess;
END_VAR

tInit(IN:= bInit, PT:= T#500MS, Q=> , ET=> );
IF NOT tInit.Q THEN
	nStep:=10;
	bInit:=TRUE;
	RETURN;
END_IF

CASE nStep OF
	0:
		;
	10:
		bDone:=FALSE;
		bErrDone:=FALSE;
		sErrTxt:='';
		fbNT_StartProcess(Start:=FALSE);
		nStep:=nStep+10;
	20:
		fbNT_StartProcess(
			NETID:= , 
			PATHSTR:= '\Windows\system32\cmd.exe', 
			DIRNAME:= '\Windows\system32', 
			COMNDLINE:= '/c services refresh htp0:', 
			START:= TRUE, 
			TMOUT:= , 
			BUSY=> , 
			ERR=> , 
			ERRID=> );
		IF NOT fbNT_StartProcess.BUSY THEN
			IF fbNT_StartProcess.ERR THEN
				sErrTxt:=CONCAT('Could not restart webserver! ErrorID: ', TO_STRING(fbNT_StartProcess.ERRID));
				bErrDone:=TRUE;
				nStep:=0;
			ELSE
				nStep:=nStep+10;
			END_IF
			fbNT_StartProcess(Start:=FALSE);
		END_IF
	30:
		nStep:=nStep+10;
	40:
		fbNT_StartProcess(Start:=FALSE);
		nStep:=nStep+10;
	50:
		fbNT_StartProcess(
			NETID:= , 
			PATHSTR:= '\Windows\system32\cmd.exe', 
			DIRNAME:= '\Windows\system32', 
			COMNDLINE:= '/c iisreset/restart', 
			START:= TRUE, 
			TMOUT:= , 
			BUSY=> , 
			ERR=> , 
			ERRID=> );
		IF NOT fbNT_StartProcess.BUSY THEN
			IF fbNT_StartProcess.ERR THEN
				sErrTxt:=CONCAT('Could not restart webserver! ErrorID: ', TO_STRING(fbNT_StartProcess.ERRID));
				bErrDone:=TRUE;
				nStep:=0;
			ELSE
				nStep:=nStep+10;
			END_IF
			fbNT_StartProcess(Start:=FALSE);
		END_IF
	60:
		nStep:=100;
	
	100:
		bDone:=TRUE;
		nStep:=0;
END_CASE

END_PROGRAM

// ---- POUs/MachinePOU/State/otherMachineState.TcPOU
PROGRAM otherMachineState
VAR_INPUT
	lightShow:BOOL;
END_VAR
VAR
	inChamberState:UDINT;
	outChamberState:UDINT;
	etchState:UDINT;
	t1:TON;
	rTrig:R_TRIG;
END_VAR

// Chamber State
// Wafer In Chamber State
IF gCtrlMode=ControlMode.eManualCtrMode THEN
	CASE inChamberState OF
		0:
			// 无 Wafer 状态
			IF gWaferMemoryState=0 THEN
				inChamberState:=inChamberState+10;
			END_IF
		10:
			// 实时检测放入晶圆
			IF gICP.I_WaferCheck AND gICP.I_ARMHome THEN
				inChamberState:=inChamberState+10;
			ELSE
				inChamberState:=0;
			END_IF
		20:
			IF gICP.GateDoorExtSensor THEN
				inChamberState:=inChamberState+10;
			ELSE
				inChamberState:=0;
			END_IF
		30:
			IF NOT gICP.I_ARMHome THEN
				inChamberState:=inChamberState+10;
			ELSE
				inChamberState:=20;
			END_IF
		40:
			IF gARMPosition=gICP.ARM.actpos THEN
				inChamberState:=inChamberState+10;
			ELSE
				inChamberState:=20;
			END_IF
		50:
			IF gICP.LiftPinExtSensor THEN// 顶起
				inChamberState:=100;
				gWaferMemoryState:=1;
				ups_CX51X0.Act_Wrtie();
			ELSE
				inChamberState:=200;// 不顶起
				gWaferMemoryState:=0;
				ups_CX51X0.Act_Wrtie();
			END_IF
		100:
			IF ABS( gARMPosition-gICP.ARM.actpos)>1 THEN// 手臂回原
				inChamberState:=inChamberState+10;
			ELSE
				inChamberState:=50;// 手臂静止
			END_IF
		110:
			IF gICP.I_ARMHome THEN
				inChamberState:=0;
			END_IF
			IF gARMPosition=gICP.ARM.actpos THEN
				inChamberState:=40;
			END_IF
		200:
			IF ABS( gARMPosition-gICP.ARM.actpos)>1 THEN// 手臂回原
				inChamberState:=inChamberState+10;
			ELSE
				inChamberState:=50;// 手臂静止
			END_IF
		210:
			IF gICP.I_ARMHome THEN
				inChamberState:=0;
			END_IF
			IF gARMPosition=gICP.ARM.actpos THEN
				inChamberState:=40;
			END_IF
	END_CASE
	
	CASE outChamberState OF
		0:
			// 有 Wafer 状态
			IF gWaferMemoryState=1 THEN
				outChamberState:=outChamberState+10;
			END_IF
		10:
			IF gICP.GateDoorExtSensor AND gARMPosition=gICP.ARM.actpos THEN
				outChamberState:=outChamberState+10;
			ELSE
				outChamberState:=0;
			END_IF
		20:
			IF gICP.LiftPinExtSensor THEN
				outChamberState:=outChamberState+10;
			END_IF
		30:
			IF gICP.LiftPinRetSensor THEN
				gWaferMemoryState:=0;
				ups_CX51X0.Act_Wrtie();
				outChamberState:=outChamberState+10;
			ELSE
				IF ABS( gARMPosition-gICP.ARM.actpos)>1 THEN
					outChamberState:=0;
				END_IF
			END_IF	
		40:
			IF gICP.I_ARMHome THEN
				outChamberState:=0;
			END_IF
			IF gICP.LiftPinExtSensor THEN
				gWaferMemoryState:=1;
				ups_CX51X0.Act_Wrtie();
				outChamberState:=20;
			END_IF
	END_CASE
END_IF
t1(IN:=gWaferMemoryState=1 AND NOT t1.Q,PT:=T#0.5S);
IF t1.Q THEN
	lightShow:=NOT lightShow;
END_IF
IF gWaferMemoryState=0 THEN
	lightShow:=FALSE;
END_IF

IF S_ActuatorRecoveryPOU.busy OR MainPOU.busy OR S_ChamberLLVent.busy OR S_Etching.busy OR S_LoadLockPumping.busy OR S_LoadLockVent.busy OR
	S_LoadWafer.busy OR S_MachinePumping.busy OR S_MachineVent.busy OR S_RoughPumping.busy OR S_UnLoadWafer.busy OR S_WaferCheckPOU.busy OR
	S_PDVSafeCtr.busy THEN
	gSPOUBusy:=TRUE;
ELSE
	gSPOUBusy:=FALSE;
	gShowPOURunLog:=FALSE;
END_IF
gRunningLog.clearShowInfo:=FALSE;
rTrig(CLK:=gSPOUBusy);
IF rTrig.Q THEN
	gRunningLog.clearShowInfo:=TRUE;
	gShowPOURunLog:=TRUE;
END_IF
IF NOT gSPOUBusy THEN
	IF gICP.TBGauge.outputValue<400 THEN
		gRoughRemainTMPCanOpen:=TRUE;
	ELSE
		gRoughRemainTMPCanOpen:=FALSE;
	END_IF
ELSE
	IF gICP.TBGauge.outputValue>400 THEN
		gRoughRemainTMPCanOpen:=FALSE;
	END_IF
END_IF

IF ABS(gICP.MFC1.setFlow-gICP.MFC1.actflow)>gMFCMonitParLimit OR  ABS(gICP.MFC2.setFlow-gICP.MFC2.actflow)>gMFCMonitParLimit OR  ABS(gICP.MFC3.setFlow-gICP.MFC3.actflow)>gMFCMonitParLimit 
	OR  ABS(gICP.MFC4.setFlow-gICP.MFC4.actflow)>gMFCMonitParLimit OR  ABS(gICP.MFC5.setFlow-gICP.MFC5.actflow)>gMFCMonitParLimit OR  ABS(gICP.MFC6.setFlow-gICP.MFC6.actflow)>gMFCMonitParLimit 
	OR  ABS(gICP.MFC7.setFlow-gICP.MFC7.actflow)>gMFCMonitParLimit OR  ABS(gICP.MFC8.setFlow-gICP.MFC8.actflow)>gMFCMonitParLimit OR  ABS(gICP.MFC9.setFlow-gICP.MFC9.actflow)>gMFCMonitParLimit  THEN
	gICP.S_MFCMonitFlowNotZero:=TRUE;
ELSE
	gICP.S_MFCMonitFlowNotZero:=FALSE;
END_IF

METHOD RecipeInputCheck : BOOL
VAR_INPUT
	numMax:INT;
END_VAR
VAR
	start:INT:=1;
	i:INT;
END_VAR
FOR start:=1 TO numMax DO
	IF len(gRecipeViewData[start].mfc1)>0 THEN
		FOR i:=0 TO LEN(gRecipeViewData[start].mfc1)-1 DO
			gLog.append(BYTE_TO_STRING(gRecipeViewData[start].mfc1[i]));
		END_FOR
	END_IF
END_FOR
END_METHOD

END_PROGRAM

// ---- POUs/MachinePOU/SemiAutomatic/S_ActuatorRecoveryPOU.TcPOU
PROGRAM S_ActuatorRecoveryPOU
VAR_INPUT
	bInit				:BOOL:=FALSE;// 初始化状态 busy/done/errDone
	bTrig				:BOOL:=FALSE;// 执行触发 信号
	bReset				:BOOL:=FALSE;// 报错 复位
	bPause				:BOOL:=FALSE;// 暂停 运行
	bStop				:BOOL:=FALSE;// 停止 运行
	bAbort				:BOOL:=FALSE;// 中止 运行
	
	atmflag:BOOL;
END_VAR
VAR_OUTPUT
	busy				:BOOL;
	done				:BOOL;
	errDone				:BOOL;
END_VAR
VAR
	actStep				:ActStepBase;
END_VAR
VAR
	i: INT;
	t1:ton;
	t2:ton;
	t3:ton;
	notchoose:BOOL;
//	str:STRING;
//	wstr:WSTRING;
END_VAR

busy:=actStep.isBusy();
done:=actStep.isDone();
errDone:=actStep.isError();
actStep.Act_Pause(pause:=bPause);

IF bTrig THEN
	bTrig:=FALSE;
	IF NOT busy THEN
		actStep.Act_ex();
	END_IF
END_IF

//状态复位
IF bInit THEN
	bInit:=FALSE;
	Act_init_status();
END_IF

IF bAbort OR bStop THEN
	bAbort:=FALSE;
	bStop:=FALSE;
	Act_init_status();
	actStep.toZeroStep();
	gShowLogTextTitle:='NON';
END_IF
ActionRun(tempActStep:=actStep);

(*
---Trigger action
*)
METHOD Act_Ex : BOOL
VAR_INPUT
END_VAR
IF NOT busy THEN
	actStep.Act_ex();
	Act_Ex:=TRUE;
ELSE
	Act_Ex:=FALSE;
END_IF
END_METHOD

(*
---功能: 状态复位 busy/done/errDone;
*)
METHOD Act_Init_Status
VAR_INPUT
END_VAR
actStep.Act_Init();
END_METHOD

METHOD PRIVATE ActionRun
VAR_INPUT
	tempActStep:ITFActStep;
END_VAR
VAR
END_VAR
VAR_STAT//此处定义静态变量, 保证每次进入该函数时能够在线监控当前值
	tempStep:DINT;
END_VAR
tempStep:=tempActStep.getStep();
CASE tempStep OF
0:
	IF tempActStep.isEx() THEN
		tempActStep.setBusyFlag();
		tempActStep.toBeginStep();
	END_IF
	t1(IN:= FALSE );
	t2(IN:= FALSE );
	t3(IN:= FALSE );
10:
	gShowLogTextTitle:='Actuator Recovery';
	IF gRunningState<>RunningStatus.eErrorState THEN
		tempActStep.addStep(5,FALSE);
		// 电源先关闭
		gICP.SourceRF.Act_Close();
		gICP.PowerRF.Act_Close();
		// 按道理先跳转去开气开水
		gRunningLog.append(CONCAT('Actuator Recovery POU Run:',DINT_TO_STRING(tempStep)));
		gRunningLog.append('Actuator Recovery POU Run: RF Close');
	ELSE
		error_Trigger(105);
		IF gCtrlMode=ControlMode.eManualCtrMode THEN
			tempActStep.toErrDoneStep();
		END_IF
	END_IF
15:// 是否需要加上超时处理？？？？？？？？？？？？
	IF gICP.SourceRF.Get_Done_Close() AND gICP.PowerRF.Get_Done_Close() THEN
		tempActStep.addStep(5,FALSE);
	END_IF
20:// 动阀前，先将手臂收回
	IF gICP.I_ARMHome THEN
		tempActStep.toStep(150,FALSE);
	ELSE
		tempActStep.toStep(100,FALSE);
	END_IF
	
100:
	IF gICP.GateDoorValve.Get_Done_Ext() THEN
		tempActStep.addStep(30,FALSE);
		gRunningLog.append(CONCAT('Actuator Recovery POU Run:',DINT_TO_STRING(tempStep)));
		gRunningLog.append('Actuator Recovery POU Run: GateDoor open Done');
	ELSE
		tempActStep.addStep(10,FALSE);
		gRunningLog.append(CONCAT('Actuator Recovery POU Run:',DINT_TO_STRING(tempStep)));
		gRunningLog.append('Actuator Recovery POU Run: GateDoor open');
	END_IF
110:
	IF gICP.GateDoorValve.Act_Extend() THEN
		tempActStep.addStep(10,FALSE);
	END_IF
120:
	IF gICP.GateDoorValve.Get_Done_Ext() THEN
		gRunningLog.append(CONCAT('Actuator Recovery POU Run:',DINT_TO_STRING(tempStep)));
		gRunningLog.append('Actuator Recovery POU Run: GateDoor open Done');
		tempActStep.addStep(10,FALSE);
		t1(IN:= FALSE );
		t2(IN:= FALSE );
		t3(IN:= FALSE );
		RETURN;
	END_IF
	t3(IN:= TRUE,PT:=T#5S );
	IF t3.Q THEN
		error_Trigger(106);
		t1(IN:= FALSE );
		t2(IN:= FALSE );
		t3(IN:= FALSE );
		RETURN;
	END_IF
130:
	IF gICP.ARM.Act_HOME_Auto() THEN
		gRunningLog.append(CONCAT('Actuator Recovery POU Run:',DINT_TO_STRING(tempStep)));
		gRunningLog.append('Actuator Recovery POU Run: ARM Homing');
		tempActStep.addStep(10,FALSE);
	END_IF
140:
	IF gICP.ARM.Get_Done_HOME() AND gICP.I_ARMHome THEN
		gRunningLog.append(CONCAT('Actuator Recovery POU Run:',DINT_TO_STRING(tempStep)));
		gRunningLog.append('Actuator Recovery POU Run: ARM Homing Done');
		tempActStep.addStep(10,FALSE);
		t1(IN:= FALSE );
		t2(IN:= FALSE );
		t3(IN:= FALSE );
		RETURN;
	END_IF
	t3(IN:= TRUE,PT:=T#20S );
	IF t3.Q THEN
		error_Trigger(106);
		tempActStep.addStep(5,FALSE);
		t1(IN:= FALSE );
		t2(IN:= FALSE );
		t3(IN:= FALSE );
		RETURN;
	END_IF
145:
	tempActStep.addStep(-15,TRUE);
150:
	tempActStep.toStep(300,FALSE);//
200:
	tempActStep.addStep(10,TRUE);
210:
	// 分三组，气柜、非气柜、摇摆阀和门阀
	IF (NOT gICP.ForlinLineValveExtRelay OR gICP.ForlinLineValve.Get_Done_Ret()) AND 
		(NOT gICP.RoughValveExtRelay OR gICP.RoughValve.Get_Done_Ret()) AND 
		(NOT gICP.FastPummingExtRelay OR gICP.FastPummingValve.Get_Done_Ret()) AND 
		(NOT gICP.SlowPummingExtRelay OR gICP.SlowPummingValve.Get_Done_Ret()) AND 
		(NOT gICP.VentExtRelay OR gICP.VentValve.Get_Done_Ret()) AND 
		(NOT gICP.AIMExtRelay OR gICP.AIMValve.Get_Done_Ret()) AND 
		(NOT gICP.ISOExtRelay OR gICP.ISOValve.Get_Done_Ret()) AND 
		gICP.PDVCloseSensor AND gICP.GateDoorRetSensor AND
		(NOT gICP.GVA10ExtRelay_Vent OR gICP.GVA10Valve_Vent.Get_Done_Ret()) AND 
		(NOT gICP.GASBoxVentExtRelay OR gICP.GASBoxVentValve.Get_Done_Ret()) AND 
		(NOT gICP.HeINExtRelay OR gICP.HeINValve.Get_Done_Ret()) AND 
		(NOT gICP.HePumExtRelay OR gICP.HePumValve.Get_Done_Ret()) AND 
		(gICP.ElectrodeCylRetSensor OR gICP.ElectrodeCyl.Get_Done_Ret()) AND
		(gICP.ElectrodeCylRetSensor OR gICP.ElectrodeCyl.Get_Done_Ret()) AND
		gICP.S_GASBOX_AllGVClose AND gICP.S_GASBOX_AllMFCClearDone THEN
		gRunningLog.append(CONCAT('Actuator Recovery POU Run:',DINT_TO_STRING(tempStep)));
		gRunningLog.append('Actuator Recovery POU Run: All Actuator Recovery Done');
		tempActStep.toStep(300,FALSE);
	ELSE
		tempActStep.addStep(1,FALSE);
	END_IF
211:
	IF gICP.HeMFC_ActFlow<0.2 AND gICP.HeCheckGaugeReal<0.1 AND NOT gICP.HeINExtRelay AND NOT gICP.HePumExtRelay THEN
		tempActStep.toStep(228,FALSE);
		gRunningLog.append(CONCAT('Actuator Recovery POU Run:',DINT_TO_STRING(tempStep)));
		gRunningLog.append('Actuator Recovery POU Run: Back of helium clear done');
	ELSE
		IF gICP.ChamberGauge.outputValue1>gLVacuumPressureChamber THEN
			atmflag:=TRUE;
			tempActStep.toStep(228,FALSE);
		ELSE
			atmflag:=FALSE;
			tempActStep.addStep(1,FALSE);
			gRunningLog.append(CONCAT('Actuator Recovery POU Run:',DINT_TO_STRING(tempStep)));
			gRunningLog.append('Actuator Recovery POU Run: Back of helium not clear');
		END_IF
	END_IF
212:
	tempActStep.addStep(1,TRUE);
213:
	IF gICP.HeINValve.Act_Retract() THEN
		tempActStep.addStep(1,FALSE);
		gRunningLog.append(CONCAT('Actuator Recovery POU Run:',DINT_TO_STRING(tempStep)));
		gRunningLog.append('Actuator Recovery POU Run: HeIN Close');
	END_IF
214:
	IF gICP.HeINValve.Get_Done_Ret() THEN
		tempActStep.addStep(1,FALSE);
		gRunningLog.append(CONCAT('Actuator Recovery POU Run:',DINT_TO_STRING(tempStep)));
		gRunningLog.append('Actuator Recovery POU Run: HeIN Close');
	END_IF
215:
	tempActStep.addStep(1,TRUE);
216:
	IF gICP.HePumValve.Act_Extend() THEN
		tempActStep.addStep(1,FALSE);
		gRunningLog.append(CONCAT('Actuator Recovery POU Run:',DINT_TO_STRING(tempStep)));
		gRunningLog.append('Actuator Recovery POU Run: HePumValve Open');
	END_IF
217:
	IF gICP.HePumValve.Get_Done_Ext() THEN
		tempActStep.addStep(1,FALSE);
		gRunningLog.append(CONCAT('Actuator Recovery POU Run:',DINT_TO_STRING(tempStep)));
		gRunningLog.append('Actuator Recovery POU Run: HePumValve Open done');
	END_IF
218:
	t2(IN:=TRUE ,PT:=T#2S);
	IF t2.Q THEN
		t1(IN:= FALSE );
		t2(IN:= FALSE );
		t3(IN:= FALSE );
		tempActStep.addStep(1,FALSE);
	END_IF
219:
	t1(IN:=gICP.HeMFC_ActFlow<0.2 AND gICP.HeCheckGaugeReal<0.1 ,PT:=T#2S);
	IF t1.Q THEN
		t1(IN:= FALSE );
		t2(IN:= FALSE );
		t3(IN:= FALSE );
		gICP.HePumValve.Act_Retract();
		gRunningLog.append(CONCAT('Actuator Recovery POU Run:',DINT_TO_STRING(tempStep)));
		gRunningLog.append('Actuator Recovery POU Run: HePumValve close');
		tempActStep.addStep(1,FALSE);
	END_IF
220:
	IF gICP.HeINValve.Act_Retract() THEN
		tempActStep.addStep(1,FALSE);
		gRunningLog.append(CONCAT('Actuator Recovery POU Run:',DINT_TO_STRING(tempStep)));
		gRunningLog.append('Actuator Recovery POU Run: HePumValve close done');
	END_IF
221:
	IF gICP.HeINValve.Get_Done_Ret() THEN
		tempActStep.addStep(1,FALSE);
	END_IF
222:
	tempActStep.addStep(1,TRUE);
223:
	IF gICP.HePumValve.Act_Extend() THEN
		tempActStep.addStep(1,FALSE);
	END_IF
224:
	IF gICP.HePumValve.Get_Done_Ext() THEN
		tempActStep.addStep(1,FALSE);
	END_IF
225:
	t2(IN:=TRUE ,PT:=T#2S);
	IF t2.Q THEN
		t1(IN:= FALSE );
		t2(IN:= FALSE );
		t3(IN:= FALSE );
		tempActStep.addStep(1,FALSE);
	END_IF
226:
	t1(IN:=gICP.HeMFC_ActFlow<0.2 AND gICP.HeCheckGaugeReal<0.1 AND gICP.ChamberGauge.outputValue1<500.0 AND NOT gICP.ChamberGauge.error,PT:=T#2S);
	IF t1.Q THEN
		t1(IN:= FALSE );
		t2(IN:= FALSE );
		t3(IN:= FALSE );
		gICP.HePumValve.Act_Retract();
		tempActStep.addStep(1,FALSE);
	END_IF
227:
	IF gICP.HePumValve.Get_Done_Ret() THEN
		tempActStep.addStep(1,FALSE);
	END_IF
228:
	IF 
	gICP.RoughValve.Act_Retract() AND 
	gICP.FastPummingValve.Act_Retract() AND
	gICP.SlowPummingValve.Act_Retract() AND
	gICP.VentValve.Act_Retract() AND
	gICP.AIMValve.Act_Retract() AND
	gICP.ISOValve.Act_Retract() AND
	gICP.GateDoorValve.Act_Retract() AND
	gICP.GVA10Valve_Vent.Act_Retract() AND
	gICP.GASBoxVentValve.Act_Retract() AND
	gICP.HeINValve.Act_Retract() AND
	gICP.HePumValve.Act_Retract() AND
	gICP.ElectrodeCyl.Act_Retract()  AND
	gICP.LiftPinCyl.Act_Retract() THEN
	IF (gRoughRemain) THEN
		tempActStep.addStep(2,FALSE);
		gRunningLog.append(CONCAT('Actuator Recovery POU Run:',DINT_TO_STRING(tempStep)));
		gRunningLog.append('Actuator Recovery POU Run: ALL Valve Recovery');
	ELSE
		IF gICP.ForlinLineValve.Act_Retract() THEN
			tempActStep.addStep(2,FALSE);
			gRunningLog.append(CONCAT('Actuator Recovery POU Run:',DINT_TO_STRING(tempStep)));
			gRunningLog.append('Actuator Recovery POU Run: ALL Valve Recovery');
		END_IF
	END_IF
	END_IF;
230:
	IF gRoughRemain THEN
		t1(IN:=	(NOT gICP.RoughValveExtRelay AND gICP.RoughValve.Get_Done_Ret()) AND 
			(NOT gICP.FastPummingExtRelay AND gICP.FastPummingValve.Get_Done_Ret()) AND 
			(NOT gICP.SlowPummingExtRelay AND gICP.SlowPummingValve.Get_Done_Ret()) AND 
			(NOT gICP.VentExtRelay AND gICP.VentValve.Get_Done_Ret()) AND 
			(NOT gICP.AIMExtRelay AND gICP.AIMValve.Get_Done_Ret()) AND 
			(NOT gICP.ISOExtRelay AND gICP.ISOValve.Get_Done_Ret()) AND 
			(gICP.GateDoorValve.Get_Done_Ret() AND gICP.GateDoorRetSensor) AND 
			(NOT gICP.GVA10ExtRelay_Vent OR gICP.GVA10Valve_Vent.Get_Done_Ret()) AND 
			(NOT gICP.GASBoxVentExtRelay AND gICP.GASBoxVentValve.Get_Done_Ret()) AND 
			(NOT gICP.HeINExtRelay AND gICP.HeINValve.Get_Done_Ret()) AND 
			(NOT gICP.HePumExtRelay AND gICP.HePumValve.Get_Done_Ret()) AND 
			(gICP.ElectrodeCylRetSensor AND gICP.ElectrodeCyl.Get_Done_Ret()) AND
			(gICP.LiftPinRetSensor AND gICP.LiftPinCyl.Get_Done_Ret()),PT:=T#1S);
	ELSE
		t1(IN:=(NOT gICP.ForlinLineValveExtRelay AND gICP.ForlinLineValve.Get_Done_Ret()) AND 
			(NOT gICP.RoughValveExtRelay AND gICP.RoughValve.Get_Done_Ret()) AND 
			(NOT gICP.FastPummingExtRelay AND gICP.FastPummingValve.Get_Done_Ret()) AND 
			(NOT gICP.SlowPummingExtRelay AND gICP.SlowPummingValve.Get_Done_Ret()) AND 
			(NOT gICP.VentExtRelay AND gICP.VentValve.Get_Done_Ret()) AND 
			(NOT gICP.AIMExtRelay AND gICP.AIMValve.Get_Done_Ret()) AND 
			(NOT gICP.ISOExtRelay AND gICP.ISOValve.Get_Done_Ret()) AND 
			(gICP.GateDoorValve.Get_Done_Ret() AND gICP.GateDoorRetSensor) AND 
			(NOT gICP.GVA10ExtRelay_Vent OR gICP.GVA10Valve_Vent.Get_Done_Ret()) AND 
			(NOT gICP.GASBoxVentExtRelay AND gICP.GASBoxVentValve.Get_Done_Ret()) AND 
			(NOT gICP.HeINExtRelay AND gICP.HeINValve.Get_Done_Ret()) AND 
			(NOT gICP.HePumExtRelay AND gICP.HePumValve.Get_Done_Ret()) AND 
			(gICP.ElectrodeCylRetSensor AND gICP.ElectrodeCyl.Get_Done_Ret()) AND
			(gICP.LiftPinRetSensor AND gICP.LiftPinCyl.Get_Done_Ret()),PT:=T#1S);	
	END_IF
	
	IF  t1.Q THEN
		t1(IN:= FALSE );
		t2(IN:= FALSE );
		t3(IN:= FALSE );
		tempActStep.addStep(10,FALSE);
		gRunningLog.append(CONCAT('Actuator Recovery POU Run:',DINT_TO_STRING(tempStep)));
		gRunningLog.append('Actuator Recovery POU Run: ALL Valve Recovery Done');
		RETURN;
	END_IF
	t3(IN:=TRUE,PT:=T#60S);
	IF t3.Q THEN
		error_Trigger(106);
		tempActStep.toStep(200,FALSE);
		t1(IN:= FALSE );
		t2(IN:= FALSE );
		t3(IN:= FALSE );
		RETURN;
	END_IF
240:
	tempActStep.toStep(400,FALSE);
300:
	tempActStep.addStep(10,TRUE);
310:
	IF gICP.S_GASBOX_AllGVClose AND gICP.S_GASBOX_AllMFCClearDone THEN
		tempActStep.toStep(200,FALSE);
	ELSE
		gICP.C_GASBOX_AllGVBClose:=TRUE;
		gRunningLog.append(CONCAT('Actuator Recovery POU Run:',DINT_TO_STRING(tempStep)));
		gRunningLog.append('Actuator Recovery POU Run: Gas BOX GVB Valve Recovery');
		tempActStep.addStep(10,FALSE);
	END_IF
320:
	t2(IN:=gICP.S_GASBOX_AllMFCClearDone,PT:=T#5S);
	IF t2.Q THEN
		t1(IN:= FALSE );
		t2(IN:= FALSE );
		t3(IN:= FALSE );
		tempActStep.addStep(10,FALSE);
	END_IF
330:
	gICP.C_GASBOX_AllGVClose:=TRUE;
	gICP.C_GASBOX_AllMFCClear:=TRUE;
	tempActStep.addStep(10,FALSE);
340:
	t1(IN:=(gICP.S_GASBOX_AllGVClose AND gICP.S_GASBOX_AllMFCClearDone),PT:=T#2S);
	IF  t1.Q THEN
		gRunningLog.append(CONCAT('Actuator Recovery POU Run:',DINT_TO_STRING(tempStep)));
		gRunningLog.append('Actuator Recovery POU Run: Gas BOX All Valve And MFC Recovery Done');
		t1(IN:= FALSE );
		t2(IN:= FALSE );
		t3(IN:= FALSE );
		tempActStep.addStep(10,FALSE);
		RETURN;
	END_IF
	t3(IN:=TRUE,PT:=T#60S);
	IF t3.Q THEN
		error_Trigger(106);
		tempActStep.toStep(300,FALSE);
		t1(IN:= FALSE );
		t2(IN:= FALSE );
		t3(IN:= FALSE );
		RETURN;
	END_IF
350:
	tempActStep.toStep(200,FALSE);
400:
	tempActStep.addStep(10,TRUE);
410:
	IF (gICP.PDVCloseSensor OR gRoughRemain) AND gICP.GateDoorRetSensor THEN 
		tempActStep.toStep(1000,FALSE);
	ELSE
		IF gICP.PDV.Act_Retract() AND gICP.GateDoorValve.Act_Retract() THEN
			gRunningLog.append(CONCAT('Actuator Recovery POU Run:',DINT_TO_STRING(tempStep)));
			gRunningLog.append('Actuator Recovery POU Run: PDV\Gate Door Recovery');
			tempActStep.addStep(10,FALSE);
		ELSE
			error_Trigger(106);
			tempActStep.addStep(-10,FALSE);
		END_IF
	END_IF
420:
	t1(IN:=(gICP.PDVCloseSensor AND gICP.GateDoorRetSensor),PT:=T#1S);
	IF  t1.Q THEN
		t1(IN:= FALSE );
		t2(IN:= FALSE );
		t3(IN:= FALSE );
		tempActStep.addStep(10,FALSE);
		RETURN;
	END_IF
	t3(IN:=TRUE,PT:=T#10S);
	IF t3.Q THEN
		error_Trigger(106);
		tempActStep.toErrDoneStep();
		t1(IN:= FALSE );
		t2(IN:= FALSE );
		t3(IN:= FALSE );
		RETURN;
	END_IF
430:
	tempActStep.toStep(1000,FALSE);
1000:
	tempActStep.toDoneStep();

60000://Done
	tempActStep.setDoneFlag();
	tempActStep.toZeroStep();
	
65000://Error
	tempActStep.setErrDoneFlag();
	tempActStep.toZeroStep();
	error_Trigger(300);
END_CASE
END_METHOD

END_PROGRAM

// ---- POUs/Other/ActBase/ActStepBase.TcPOU
(*
---Control step base interface
*)
FUNCTION_BLOCK ActStepBase IMPLEMENTS ITFActStep
VAR CONSTANT
	{attribute 'hide'}
	BEGIN_STEP		:DINT:=10;
	{attribute 'hide'}
	DONE_STEP		:DINT:=60000;
	{attribute 'hide'}
	ERR_DONE_STEP	:DINT:=65000;
	{attribute 'hide'}
	PAUSE_STEP		:DINT:=65500;
END_VAR
VAR_INPUT
END_VAR
VAR_OUTPUT
	step			:DINT;
	errStep			:DINT;
	pauseNextStep	:DINT;
END_VAR
VAR
	//{attribute 'hide'}
	actState		:ST_ActStep_State;
END_VAR

getStep();

(*
---Continue action
*)
METHOD Act_Continue : BOOL
VAR_INPUT
END_VAR
actState.paused:=FALSE;
actState.step:=actState.nextStep;
END_METHOD

(*
---Trigger action
*)
METHOD Act_Ex : BOOL
VAR_INPUT
END_VAR
IF NOT actState.busy AND NOT actState.error THEN
	Act_Ex:=actState.ex:=actState.busy:=TRUE;
ELSE
	Act_Ex:=FALSE;
END_IF
END_METHOD

(*
---Init all status
*)
METHOD Act_Init : BOOL
VAR_INPUT
END_VAR
actState.ex:=actState.pause:=actState.busy:=actState.done:=actState.error:=FALSE;
actState.step:=actState.errStep:=step:=0;
actState.errID:=0;
actState.errMsg:='';

Act_Init:=TRUE;
END_METHOD

(*
---Pause action
*)
METHOD Act_Pause : BOOL
VAR_INPUT
	pause:BOOL;
END_VAR
actState.pause:=pause;
Act_Pause:=TRUE;
END_METHOD

(*
---: add step;
---:
	nextStep: step 增量值;
	checkPause: 是否检测当前 pause; 如果 checkPause:=TRUE, 且暂停被触发后, 当前 step 暂停递增;
*)
METHOD addStep : DINT
VAR_INPUT
	nextStep			:DINT:=0;
	checkPause			:BOOL:=FALSE;// 检查是否暂停，暂停则不递增step
END_VAR
IF checkPause THEN
	IF NOT actState.pause THEN
		actState.step:=actState.step+nextStep;
	END_IF
ELSE
	actState.step:=actState.step+nextStep;
END_IF

addStep:=step:=actState.step;
END_METHOD

(*
---Get action state
*)
METHOD getActState : ST_ActStep_State
VAR_INPUT
END_VAR
getActState:=actState;
END_METHOD

(*
---Get error id
*)
METHOD getErrID : DINT
VAR_INPUT
END_VAR
getErrID:=actState.errID;
END_METHOD

(*
---Get error message
*)
METHOD getErrMsg : STRING(255)
VAR_INPUT
END_VAR
getErrMsg:=actState.errMsg;
END_METHOD

(*
---Get error step
*)
METHOD getErrStep : DINT
VAR_INPUT
END_VAR
getErrStep:=actState.errStep;
END_METHOD

(*
---Get step
*)
METHOD getStep : DINT
VAR_INPUT
END_VAR
getStep:=step:=actState.step;
END_METHOD

(*
---Check busy state
*)
METHOD isBusy : BOOL
VAR_INPUT
END_VAR

isBusy:=actState.busy;
END_METHOD

(*
---Check done state
*)
METHOD isDone : BOOL
VAR_INPUT
END_VAR

isDone:=actState.done;
END_METHOD

(*
---Check error state
*)
METHOD isError : BOOL
VAR_INPUT
END_VAR

isError:=actState.error;
END_METHOD

(*
---Check trigger state
*)
METHOD isEx : BOOL
VAR_INPUT
END_VAR

isEx:=actState.ex;
END_METHOD

(*
---Check pause state
*)
METHOD isPause : BOOL
VAR_INPUT
END_VAR

isPause:=actState.pause;
END_METHOD

(*
---Set busy flag
*)
METHOD setBusyFlag
VAR_INPUT
END_VAR
//actState.busy:=TRUE;
actState.ex:=actState.done:=actState.error:=FALSE;
actState.errID:=0;
actState.step:=step:=actState.errStep:=errStep:=actState.nextStep:=pauseNextStep:=0;
actState.errMsg:='';
END_METHOD

(*
---Set done flag
*)
METHOD setDoneFlag
VAR_INPUT
END_VAR
actState.busy:=FALSE;
actState.pause:=FALSE;
actState.done:=TRUE;
actState.error:=FALSE;
actState.errID:=0;
actState.errMsg:='';
END_METHOD

(*
---Set error done flag
*)
METHOD setErrDoneFlag
VAR_INPUT
END_VAR
actState.busy:=FALSE;
actState.pause:=FALSE;
actState.done:=FALSE;
actState.error:=TRUE;
END_METHOD

(*
---Set error id
*)
METHOD setErrID
VAR_INPUT
	errID:DINT;
END_VAR
actState.errID:=errID;
errStep:=actState.errStep:=actState.step;
END_METHOD

(*
---Set error message
*)
METHOD setErrMsg
VAR_INPUT
	errMsg:STRING(255);
END_VAR
actState.errMsg:=errMsg;
errStep:=actState.errStep:=actState.step;
END_METHOD

(*
---Set error id and error message
*)
METHOD setError
VAR_INPUT
	errID:DINT;
	errMsg:STRING(255);
END_VAR
setErrID(errID);
setErrMsg(errMsg);
END_METHOD

(*
---Go to step:=BEGIN_STEP, BEGIN_STEP is 10;
*)
METHOD toBeginStep : DINT
VAR_INPUT
END_VAR
toBeginStep:=step:=actState.step:=BEGIN_STEP;
END_METHOD

(*
---Go to step:=DONE_STEP, DONE_STEP is 60000;
*)
METHOD toDoneStep : DINT
VAR_INPUT
END_VAR
toDoneStep:=step:=actState.step:=DONE_STEP;
END_METHOD

(*
---Go to step:=ERR_DONE_STEP, ERR_DONE_STEP is 65000;
*)
METHOD toErrDoneStep : DINT
VAR_INPUT
END_VAR
errStep:=actState.errStep:=actState.step;
toErrDoneStep:=step:=actState.step:=ERR_DONE_STEP;
END_METHOD

(*
---Go to pause step:=PAUSE_STEP, PAUSE_STEP is 65500; 
---: nextStep: 从暂停解除之后的下一个step值; 
*)
METHOD toPauseStep : DINT
VAR_INPUT
	nextStep			:DINT:=0;
END_VAR
actState.paused:=TRUE;
actState.nextStep:=pauseNextStep:=nextStep;
actState.step:=PAUSE_STEP;
END_METHOD

(*
---: Go to target step;
---:
	nextStep: step 目标值;
	checkPause: 是否检测当前 pause; 如果 checkPause:=TRUE, 且暂停被触发后, 当前 step 暂停递增;
*)
METHOD toStep : DINT
VAR_INPUT
	nextStep			:DINT:=0;// 跳转到目标step
	checkPause			:BOOL:=FALSE;// 检查是否暂停，暂停则不递增step
END_VAR
IF checkPause THEN
	IF NOT actState.pause THEN
		actState.step:=nextStep;
	END_IF
ELSE
	actState.step:=nextStep;
END_IF

toStep:=step:=actState.step;
END_METHOD

(*
---Go to step:=0;
*)
METHOD toZeroStep : DINT
VAR_INPUT
END_VAR
toZeroStep:=step:=actState.step:=0;
END_METHOD

END_FUNCTION_BLOCK

// ---- POUs/MachinePOU/MainPOU.TcPOU
PROGRAM MainPOU
VAR_INPUT
	bInit				:BOOL:=FALSE;// 初始化状态 busy/done/errDone
	bTrig				:BOOL:=FALSE;// 执行触发 信号
	bReset				:BOOL:=FALSE;// 报错 复位
	bPause				:BOOL:=FALSE;// 暂停 运行
	bStop				:BOOL:=FALSE;// 停止 运行
	bAbort				:BOOL:=FALSE;// 中止 运行
	
	DUTCount			:INT:=1;
	showmsg				:BOOL;//弹窗确认模式
	swcomfirmButton		:BOOL;
END_VAR
VAR_OUTPUT
	busy				:BOOL;
	done				:BOOL;
	errDone				:BOOL;
END_VAR
VAR
	actStep				:ActStepBase;
END_VAR
VAR
	i: INT;
	t1:ton;
	t2:ton;
	t3:ton;
	notchoose:BOOL;
END_VAR

busy:=actStep.isBusy();
done:=actStep.isDone();
errDone:=actStep.isError();
actStep.Act_Pause(pause:=bPause);

IF bTrig THEN
	bTrig:=FALSE;
	IF NOT busy THEN
		actStep.Act_ex();
	END_IF
END_IF

//状态复位
IF bInit THEN
	bInit:=FALSE;
	Act_init_status();
	showmsg:=FALSE;
END_IF

IF bAbort OR bStop THEN
	bAbort:=FALSE;
	bStop:=FALSE;
	Act_init_status();
	actStep.toZeroStep();
	showmsg:=FALSE;
END_IF
ActionRun(tempActStep:=actStep);

(*
---Trigger action
*)
METHOD Act_Ex : BOOL
VAR_INPUT
END_VAR
IF NOT busy THEN
	actStep.Act_ex();
	Act_Ex:=TRUE;
ELSE
	Act_Ex:=FALSE;
END_IF
END_METHOD

(*
---功能: 状态复位 busy/done/errDone;
*)
METHOD Act_Init_Status
VAR_INPUT
END_VAR
actStep.Act_Init();
END_METHOD

METHOD PRIVATE ActionRun
VAR_INPUT
	tempActStep:ITFActStep;
END_VAR
VAR
END_VAR
VAR_STAT//此处定义静态变量, 保证每次进入该函数时能够在线监控当前值
	tempStep:DINT;
END_VAR
tempStep:=tempActStep.getStep();
CASE tempStep OF
0:
	IF tempActStep.isEx() THEN
		tempActStep.setBusyFlag();
		tempActStep.toBeginStep();
	END_IF
	t1(IN:= FALSE );
	t2(IN:= FALSE );
	t3(IN:= FALSE );
10:
	IF gWaferMemoryState=2 THEN
		tempActStep.toStep(300,FALSE);// UnLoad
	ELSIF gWaferMemoryState=1 THEN
		tempActStep.toStep(200,FALSE);// Etching
	ELSIF gWaferMemoryState=0 THEN	
		tempActStep.toStep(100,FALSE);// Load
	END_IF
100:
	tempActStep.addStep(10,TRUE);
110:
	S_LoadWafer.Act_Init_Status();
	S_LoadWafer.Act_Ex();
	tempActStep.addStep(10,FALSE);
120:
	IF S_LoadWafer.busy THEN
		tempActStep.addStep(10,FALSE);
	END_IF
130:
	IF S_LoadWafer.done THEN
		tempActStep.addStep(10,FALSE);
		RETURN;
	END_IF
	IF S_LoadWafer.errDone THEN
		tempActStep.toErrDoneStep();
		RETURN;
	END_IF
140:
	tempActStep.toStep(10,FALSE);
	
200:
	tempActStep.addStep(10,TRUE);
210:
	S_Etching.Act_Init_Status();
	S_Etching.Act_Ex();
	tempActStep.addStep(10,FALSE);
220:
	IF S_Etching.busy THEN
		tempActStep.addStep(10,FALSE);
	END_IF
230:
	IF S_Etching.done THEN
		tempActStep.addStep(10,FALSE);
		RETURN;
	END_IF
	IF S_Etching.errDone THEN
		tempActStep.toErrDoneStep();
		RETURN;
	END_IF
240:
	tempActStep.toStep(10,FALSE);
	
300:
	tempActStep.addStep(10,TRUE);
310:
	S_UnLoadWafer.Act_Init_Status();
	S_UnLoadWafer.Act_Ex();
	tempActStep.addStep(10,FALSE);
320:
	IF S_UnLoadWafer.busy THEN
		tempActStep.addStep(10,FALSE);
	END_IF
330:
	IF S_UnLoadWafer.done THEN
		tempActStep.addStep(10,FALSE);
		RETURN;
	END_IF
	IF S_UnLoadWafer.errDone THEN
		tempActStep.toErrDoneStep();
		RETURN;
	END_IF
340:
	tempActStep.toStep(10,FALSE);
	
1000:
	tempActStep.toDoneStep();

60000://Done
	tempActStep.setDoneFlag();
	tempActStep.toZeroStep();
	
65000://Error
	tempActStep.setErrDoneFlag();
	tempActStep.toZeroStep();
END_CASE
END_METHOD

END_PROGRAM

// ---- POUs/MachinePOU/SemiAutomatic/S_LoadWafer.TcPOU
PROGRAM S_LoadWafer
VAR_INPUT
	bInit				:BOOL:=FALSE;// 初始化状态 busy/done/errDone
	bTrig				:BOOL:=FALSE;// 执行触发 信号
	bReset				:BOOL:=FALSE;// 报错 复位
	bPause				:BOOL:=FALSE;// 暂停 运行
	bStop				:BOOL:=FALSE;// 停止 运行
	bAbort				:BOOL:=FALSE;// 中止 运行
	
END_VAR
VAR_OUTPUT
	busy				:BOOL;
	done				:BOOL;
	errDone				:BOOL;
END_VAR
VAR
	actStep				:ActStepBase;
END_VAR
VAR
	i: INT;
	t1:ton;
	t2:ton;
	t3:ton;
	notchoose:BOOL;
	timeOutTime:TIME:= T#60S;
	ventTime:TIME:=T#20S;
END_VAR

busy:=actStep.isBusy();
done:=actStep.isDone();
errDone:=actStep.isError();
actStep.Act_Pause(pause:=bPause);

IF bTrig THEN
	bTrig:=FALSE;
	IF NOT busy THEN
		actStep.Act_ex();
	END_IF
END_IF

//状态复位
IF bInit THEN
	bInit:=FALSE;
	Act_init_status();
END_IF

IF bAbort OR bStop THEN
	bAbort:=FALSE;
	bStop:=FALSE;
	Act_init_status();
	actStep.toZeroStep();
	gShowLogTextTitle:='NON';
END_IF
ActionRun(tempActStep:=actStep);

(*
---Trigger action
*)
METHOD Act_Ex : BOOL
VAR_INPUT
END_VAR
IF NOT busy THEN
	actStep.Act_ex();
	Act_Ex:=TRUE;
ELSE
	Act_Ex:=FALSE;
END_IF
END_METHOD

(*
---功能: 状态复位 busy/done/errDone;
*)
METHOD Act_Init_Status
VAR_INPUT
END_VAR
actStep.Act_Init();
END_METHOD

METHOD PRIVATE ActionRun
VAR_INPUT
	tempActStep:ITFActStep;
END_VAR
VAR_STAT//此处定义静态变量, 保证每次进入该函数时能够在线监控当前值
	tempStep:DINT;
END_VAR
tempStep:=tempActStep.getStep();
CASE tempStep OF
0:
	IF tempActStep.isEx() THEN
		tempActStep.setBusyFlag();
		tempActStep.toBeginStep();
	END_IF
	t1(IN:= FALSE );
	t2(IN:= FALSE );
	t3(IN:= FALSE );
10:
	gShowLogTextTitle:='Load Wafer';
	IF gRunningState<>RunningStatus.eErrorState THEN
		tempActStep.addStep(10,FALSE);
	ELSE
		error_Trigger(105);
		IF gCtrlMode=ControlMode.eManualCtrMode THEN
			tempActStep.toErrDoneStep();
		END_IF
	END_IF
20:
	IF ControlMode.eManualCtrMode=gCtrlMode THEN
//		S_WaferCheckPOU.Act_Init_Status();
//		S_WaferCheckPOU.Act_Ex();
		tempActStep.addStep(10,FALSE);
	ELSIF( ControlMode.eAutoCtrMode=gCtrlMode) THEN
		tempActStep.addStep(10,FALSE);
	ELSE
		tempActStep.toErrDoneStep();
	END_IF
30:
	tempActStep.addStep(10,FALSE);
40:
	tempActStep.addStep(10,TRUE);
50:
	tempActStep.addStep(10,FALSE);
60:
	S_RoughPumping.Act_Init_Status();
	S_RoughPumping.Act_Ex();
	tempActStep.addStep(10,FALSE);
70:
	IF S_RoughPumping.done THEN
		gShowLogTextTitle:='Load Wafer';
		tempActStep.addStep(10,FALSE);
	END_IF
	IF S_RoughPumping.errDone THEN
		tempActStep.toStep(40,FALSE);
	END_IF
80:
	tempActStep.addStep(20,TRUE);
100:
	IF gWaferMemoryState=1 THEN// 腔体有晶圆
		gRunningLog.append(CONCAT('Load Wafer POU Run:',DINT_TO_STRING(tempStep)));
		gRunningLog.append('Load Wafer POU Run: Wafer In Chamber ');
		tempActStep.toStep(590,FALSE);
	ELSE// 腔体无晶圆
		gRunningLog.append(CONCAT('Load Wafer POU Run:',DINT_TO_STRING(tempStep)));
		gRunningLog.append('Load Wafer POU Run: Wafer OutSide Chamber ');
		IF NOT gICP.I_WaferCheck THEN
			tempActStep.addStep(10,FALSE);// 手臂上无晶圆
			gRunningLog.append('Load Wafer POU Run: There are wafers on the arm ');
		ELSE
			gRunningLog.append('Load Wafer POU Run: There are not wafers on the arm ');
			tempActStep.toStep(200,FALSE);// 手臂上有晶圆
		END_IF
	END_IF
110:
	tempActStep.addStep(5,TRUE);
115:
	IF  gICP.GateDoorValve.Act_Retract() AND 
	    gICP.SlowPummingValve.Act_Retract() AND 
	    gICP.FastPummingValve.Act_Retract() THEN
		gRunningLog.append(CONCAT('Load Wafer POU Run:',DINT_TO_STRING(tempStep)));
		gRunningLog.append('Load Wafer POU Run:LoadLock Close');
		tempActStep.addStep(5,FALSE);
	END_IF
120:
	IF gICP.GateDoorValve.Get_Done_Ret() AND gICP.GateDoorRetSensor AND
	   gICP.SlowPummingValve.Get_Done_Ret() AND NOT gICP.SlowPummingExtRelay AND
	   gICP.FastPummingValve.Get_Done_Ret() AND NOT gICP.FastPummingExtRelay THEN
	   gRunningLog.append(CONCAT('Load Wafer POU Run:',DINT_TO_STRING(tempStep)));
	   gRunningLog.append('Load Wafer POU Run:LoadLock Close Done');
		tempActStep.addStep(10,FALSE);
	END_IF
130:
	IF gICP.VentValve.Act_Extend() THEN
		gRunningLog.append(CONCAT('Load Wafer POU Run:',DINT_TO_STRING(tempStep)));
		gRunningLog.append('Load Wafer POU Run:Vent Open');
		tempActStep.addStep(10,FALSE);
	END_IF
140:
	IF gICP.VentValve.Get_Done_Ext() THEN
		gRunningLog.append(CONCAT('Load Wafer POU Run:',DINT_TO_STRING(tempStep)));
		gRunningLog.append('Load Wafer POU Run:Vent Open Done');
		tempActStep.addStep(10,FALSE);
	END_IF
150:
	t2(IN:=gICP.LoadLockGauge.outputValue>gATMPressure,PT:=ventTime);
	IF t2.Q OR NOT gICP.I_LLSwitch THEN
		gRunningLog.append(CONCAT('Load Wafer POU Run:',DINT_TO_STRING(tempStep)));
		gRunningLog.append(CONCAT('Load Wafer POU Run:LL Vent Pressure Arrive：',REAL_TO_STRING(gICP.LoadLockGauge.outputValue)));
		t1(IN:= FALSE );
		t2(IN:= FALSE );
		t3(IN:= FALSE );
		tempActStep.addStep(10,FALSE);
		RETURN;
	END_IF
	t1(IN:= TRUE,PT:=timeOutTime );
	IF t1.Q THEN
		t1(IN:= FALSE );
		t2(IN:= FALSE );
		t3(IN:= FALSE );
		error_Trigger(110);
		tempActStep.toStep(110,FALSE);
		RETURN;
	END_IF
160:
	tempActStep.addStep(10,TRUE);
170:
	IF gICP.VentValve.Act_Retract() THEN
		gRunningLog.append(CONCAT('Load Wafer POU Run:',DINT_TO_STRING(tempStep)));
		gRunningLog.append('Load Wafer POU Run:Vent Close');
		tempActStep.addStep(10,FALSE);
	END_IF
180:
	IF gICP.GateDoorValve.Get_Done_Ret() THEN
		gRunningLog.append(CONCAT('Load Wafer POU Run:',DINT_TO_STRING(tempStep)));
		gRunningLog.append('Load Wafer POU Run:Vent Close Done');
		tempActStep.addStep(10,FALSE);
	END_IF
190:
	t1(IN:=TRUE,PT:=T#1S);
	IF t1.Q THEN
		t1(IN:= FALSE );
		t2(IN:= FALSE );
		t3(IN:= FALSE );
		gRunningLog.append(CONCAT('Load Wafer POU Run:',DINT_TO_STRING(tempStep)));
		gRunningLog.append('Load Wafer POU Run:Wait for the wafer to be placed');
		tempActStep.addStep(10,FALSE);
	END_IF
200:
	t2(IN:=gICP.I_WaferCheck AND gICP.I_LLSwitch,PT:=T#5S);// 放入晶圆，且关上盖子
	IF t2.Q THEN
		gRunningLog.append('Load Wafer POU Run:Place the wafer and close the lid');
		t1(IN:= FALSE );
		t2(IN:= FALSE );
		t3(IN:= FALSE );
		tempActStep.addStep(10,FALSE);
		RETURN;
	END_IF
	t3(IN:=TRUE,PT:=timeOutTime);
	IF t3.Q THEN
		error_Trigger(110);
		t1(IN:= FALSE );
		t2(IN:= FALSE );
		t3(IN:= FALSE );
		tempActStep.tostep(160,FALSE);
	END_IF
210:
	tempActStep.addStep(5,TRUE);
215:
	t2(IN:=gICP.LoadLockGauge.outputValue<gRoughtPumVaccum,PT:=T#2S);
	IF t2.Q THEN
		gRunningLog.append(CONCAT('Load Wafer POU Run:',DINT_TO_STRING(tempStep)));
		gRunningLog.append(CONCAT('Load Wafer POU Run:LL Pumping Pressure Arrive：',REAL_TO_STRING(gICP.LoadLockGauge.outputValue)));
		t1(IN:= FALSE );
		t2(IN:= FALSE );
		t3(IN:= FALSE );
		tempActStep.tostep(310,FALSE);
		RETURN;
	END_IF
	t3(IN:=TRUE,PT:=T#3S);
	IF t3.Q THEN
		t1(IN:= FALSE );
		t2(IN:= FALSE );
		t3(IN:= FALSE );
		IF  gICP.VentValve.Act_Retract() AND 
			gICP.ForlinLineValve.Act_Retract() AND 
			gICP.RoughValve.Act_Retract() THEN
			gRunningLog.append(CONCAT('Load Wafer POU Run:',DINT_TO_STRING(tempStep)));
			gRunningLog.append('Load Wafer POU Run:LL Pumping(Close Vent\Forline\Rough Valve)');
			tempActStep.addStep(5,FALSE);
		END_IF
	END_IF
220:
	IF gICP.VentValve.Get_Done_Ret() AND NOT gICP.VentExtRelay AND
	   gICP.ForlinLineValve.Get_Done_Ret() AND NOT gICP.ForlinLineValveExtRelay AND
	   gICP.RoughValve.Get_Done_Ret() AND NOT gICP.RoughValveExtRelay THEN
	   gRunningLog.append(CONCAT('Load Wafer POU Run:',DINT_TO_STRING(tempStep)));
	   gRunningLog.append('Load Wafer POU Run:LL Pumping(Vent\Forline\Rough Valve Close Done)');
		tempActStep.addStep(10,FALSE);
	END_IF
230://////////////准备抽LoadLock
	tempActStep.addStep(10,FALSE);
240:
	tempActStep.addStep(10,TRUE);
250:
	IF gICP.SlowPummingValve.Act_Extend() AND gICP.FastPummingValve.Act_Retract() THEN
		gRunningLog.append(CONCAT('Load Wafer POU Run:',DINT_TO_STRING(tempStep)));
		gRunningLog.append('Load Wafer POU Run:LL Rough Pumping(SlowPum Valve Open \ FastPum Valve Close)');
		tempActStep.addStep(10,FALSE);
	END_IF
260:
	IF gICP.SlowPummingValve.Get_Done_Ext() AND gICP.FastPummingValve.Get_Done_Ret() THEN
		gRunningLog.append(CONCAT('Load Wafer POU Run:',DINT_TO_STRING(tempStep)));
		gRunningLog.append('Load Wafer POU Run:LL Rough Pumping(SlowPum Valve Open Done\ FastPum Valve Close Done)');
		tempActStep.addStep(10,FALSE);
	END_IF
270:
	t2(IN:=gICP.LoadLockGauge.outputValue<gLoadLockPumSVaccum,PT:=T#2S);
	IF t2.Q THEN
		gRunningLog.append(CONCAT('Load Wafer POU Run:',DINT_TO_STRING(tempStep)));
		gRunningLog.append(CONCAT('Load Wafer POU Run:LL Rough Pumping Pressure Arrive：',REAL_TO_STRING(gICP.LoadLockGauge.outputValue)));
		t1(IN:= FALSE );
		t2(IN:= FALSE );
		t3(IN:= FALSE );
		tempActStep.addStep(10,FALSE);
	END_IF
280:
	IF gICP.SlowPummingValve.Act_Retract() AND gICP.FastPummingValve.Act_Extend() THEN
		gRunningLog.append(CONCAT('Load Wafer POU Run:',DINT_TO_STRING(tempStep)));
		gRunningLog.append('Load Wafer POU Run:LL Fast Pumping(SlowPum Valve Close \ FastPum Valve Open)');
		tempActStep.addStep(10,FALSE);
	END_IF
290:
	IF gICP.SlowPummingValve.Get_Done_Ret() AND gICP.FastPummingValve.Get_Done_Ext() THEN
		gRunningLog.append(CONCAT('Load Wafer POU Run:',DINT_TO_STRING(tempStep)));
		gRunningLog.append('Load Wafer POU Run:LL Fast Pumping(SlowPum Valve Close Done\ FastPum Valve Open Done)');
		tempActStep.addStep(10,FALSE);
	END_IF
300:
	t2(IN:=gICP.LoadLockGauge.outputValue<gRoughtPumVaccum,PT:=T#2S);
	IF t2.Q THEN
		gRunningLog.append(CONCAT('Load Wafer POU Run:',DINT_TO_STRING(tempStep)));
		gRunningLog.append(CONCAT('Load Wafer POU Run:LL Fast Pumping Pressure Arrive：',REAL_TO_STRING(gICP.LoadLockGauge.outputValue)));
		t1(IN:= FALSE );
		t2(IN:= FALSE );
		t3(IN:= FALSE );
		tempActStep.addStep(10,FALSE);
	END_IF
310:
	tempActStep.addStep(10,TRUE);
320:
	IF gICP.SlowPummingValve.Act_Retract() AND gICP.FastPummingValve.Act_Retract() THEN
		gRunningLog.append(CONCAT('Load Wafer POU Run:',DINT_TO_STRING(tempStep)));
		gRunningLog.append('Load Wafer POU Run:LL Fast Pumping(SlowPum Valve Close \ FastPum Valve Close)');
		tempActStep.addStep(10,FALSE);
	END_IF
330:
	IF gICP.SlowPummingValve.Get_Done_Ret() AND gICP.FastPummingValve.Get_Done_Ret() THEN
		gRunningLog.append(CONCAT('Load Wafer POU Run:',DINT_TO_STRING(tempStep)));
		gRunningLog.append('Load Wafer POU Run:LL Fast Pumping(SlowPum Valve Close Done\ FastPum Valve Close Done)');
		tempActStep.addStep(10,FALSE);
	END_IF
340:
	tempActStep.addStep(2,TRUE);
342:
	IF gICP.PDV.Act_Retract() THEN
		gRunningLog.append(CONCAT('Load Wafer POU Run:',DINT_TO_STRING(tempStep)));
		gRunningLog.append('Load Wafer POU Run:PDV Close');
		tempActStep.addStep(2,FALSE);
	END_IF
344:
	IF gICP.PDV.Get_Done_Ret() OR gICP.PDVCloseSensor THEN
		gRunningLog.append(CONCAT('Load Wafer POU Run:',DINT_TO_STRING(tempStep)));
		gRunningLog.append('Load Wafer POU Run:PDV Close Done');
		tempActStep.addStep(2,FALSE);
	END_IF
346:
	tempActStep.addStep(4,TRUE);
350:
	IF gICP.GateDoorValve.Act_Extend() THEN
		gRunningLog.append(CONCAT('Load Wafer POU Run:',DINT_TO_STRING(tempStep)));
		gRunningLog.append('Load Wafer POU Run:Gate Door Open');
		tempActStep.addStep(10,FALSE);
	END_IF
360:
	IF gICP.GateDoorValve.Get_Done_Ext() AND gICP.GateDoorExtSensor THEN
		gRunningLog.append(CONCAT('Load Wafer POU Run:',DINT_TO_STRING(tempStep)));
		gRunningLog.append('Load Wafer POU Run:Gate Door Open Done');
		tempActStep.addStep(10,FALSE);
	END_IF
370:
	IF gICP.ElectrodeCyl.Act_Retract() AND gICP.LiftPinCyl.Act_Retract() THEN
		gRunningLog.append(CONCAT('Load Wafer POU Run:',DINT_TO_STRING(tempStep)));
		gRunningLog.append('Load Wafer POU Run:ElectrodeCyl&LiftPinCyl Down');
		tempActStep.addStep(10,FALSE);
	END_IF
380:
	IF gICP.ElectrodeCyl.Get_Done_Ret() AND gICP.LiftPinCyl.Get_Done_Ret() THEN
		gRunningLog.append(CONCAT('Load Wafer POU Run:',DINT_TO_STRING(tempStep)));
		gRunningLog.append('Load Wafer POU Run:ElectrodeCyl&LiftPinCyl Down Done');
		tempActStep.addStep(10,FALSE);
	END_IF
390:
	tempActStep.addStep(10,TRUE);
400:
	IF gICP.ARM.Act_IN_Auto() THEN
		gRunningLog.append(CONCAT('Load Wafer POU Run:',DINT_TO_STRING(tempStep)));
		gRunningLog.append('Load Wafer POU Run:ARM IN');
		tempActStep.addStep(10,FALSE);
	END_IF
410:
	IF NOT gICP.I_ARMHome THEN// 手臂当前不应该在原点位置
		gRunningLog.append(CONCAT('Load Wafer POU Run:',DINT_TO_STRING(tempStep)));
		gRunningLog.append('Load Wafer POU Run:ARM Running');
		tempActStep.addStep(10,FALSE);
	END_IF
420:
	t2(IN:=gICP.ARM.Get_Done_IN() AND NOT(gICP.ARM.busy OR gICP.ARM.jogBusy),PT:=T#3S);
	IF t2.Q  THEN
		t1(IN:= FALSE );
		t2(IN:= FALSE );
		t3(IN:= FALSE );
		gRunningLog.append(CONCAT('Load Wafer POU Run:',DINT_TO_STRING(tempStep)));
		gRunningLog.append('Load Wafer POU Run:ARM IN Done');
		tempActStep.addStep(10,FALSE);
		RETURN;
	END_IF
	t1(IN:=TRUE,PT:=T#30S);
	IF t1.Q THEN
		t1(IN:= FALSE );
		t2(IN:= FALSE );
		t3(IN:= FALSE );
		error_Trigger(111);
		tempActStep.toStep(390,FALSE);// 报错
		RETURN;
	END_IF
430:
	tempActStep.addStep(10,TRUE);
440:
	IF gICP.LiftPinCyl.Act_Extend() THEN
		tempActStep.addStep(10,FALSE);
	END_IF
450:
	IF gICP.LiftPinCyl.Get_Done_Ext() AND gICP.LiftPinExtSensor THEN
		gRunningLog.append(CONCAT('Load Wafer POU Run:',DINT_TO_STRING(tempStep)));
		gRunningLog.append('Load Wafer POU Run:LiftPinCyl UP And Remember Wafer Memory ');
		// 记忆状态更新
		gWaferMemoryState:=1;
		ups_CX51X0.Act_Wrtie();
		tempActStep.addStep(10,FALSE);
	END_IF
460:
	tempActStep.addStep(10,TRUE);
470:
	IF gICP.ARM.Act_HOME_Auto() THEN
		gRunningLog.append(CONCAT('Load Wafer POU Run:',DINT_TO_STRING(tempStep)));
		gRunningLog.append('Load Wafer POU Run:ARM Home ');
		tempActStep.addStep(10,FALSE);
	END_IF
480:
	IF gICP.ARM.Get_Done_HOME() AND gICP.I_ARMHome AND NOT(gICP.ARM.busy OR gICP.ARM.jogBusy) THEN// 手臂当前不应该在原点位置
		gRunningLog.append(CONCAT('Load Wafer POU Run:',DINT_TO_STRING(tempStep)));
		gRunningLog.append('Load Wafer POU Run:ARM Home Done');
		tempActStep.addStep(10,FALSE);
	END_IF
490:
	t2(IN:=TRUE,PT:=T#3S);
	IF t2.Q THEN
		t1(IN:= FALSE );
		t2(IN:= FALSE );
		t3(IN:= FALSE );
		tempActStep.addStep(10,FALSE);
		RETURN;
	END_IF
500:
	tempActStep.addStep(10,TRUE);
510:
	IF gICP.GateDoorValve.Act_Retract() AND gICP.LiftPinCyl.Act_Retract() THEN
		gRunningLog.append(CONCAT('Load Wafer POU Run:',DINT_TO_STRING(tempStep)));
		gRunningLog.append('Load Wafer POU Run:Gate Door Close And LiftPinCyl Down');
		tempActStep.addStep(10,FALSE);
	END_IF
520:
	IF gICP.GateDoorValve.Get_Done_Ret() AND gICP.GateDoorRetSensor AND
	   gICP.LiftPinCyl.Get_Done_Ret() AND gICP.LiftPinRetSensor THEN
	   gRunningLog.append(CONCAT('Load Wafer POU Run:',DINT_TO_STRING(tempStep)));
	   gRunningLog.append('Load Wafer POU Run:Gate Door Close Done And LiftPinCyl Down Done');
		tempActStep.addStep(10,FALSE);
	END_IF
530:
	tempActStep.addStep(10,TRUE);
540:
	IF gICP.ForlinLineValve.Act_Extend() THEN
		gRunningLog.append(CONCAT('Load Wafer POU Run:',DINT_TO_STRING(tempStep)));
		gRunningLog.append('Load Wafer POU Run:ForLine Valve Open');
		tempActStep.addStep(10,FALSE);
	END_IF
550:
	IF gICP.ForlinLineValve.Get_Done_Ext() THEN
		gRunningLog.append(CONCAT('Load Wafer POU Run:',DINT_TO_STRING(tempStep)));
		gRunningLog.append('Load Wafer POU Run:ForLine Valve Open Done');
		tempActStep.addStep(10,FALSE);
	END_IF
560:
	tempActStep.addStep(10,TRUE);
570:
	IF gICP.PDV.Act_Open() THEN
		gRunningLog.append(CONCAT('Load Wafer POU Run:',DINT_TO_STRING(tempStep)));
		gRunningLog.append('Load Wafer POU Run:PDV Open');
		tempActStep.addStep(10,FALSE);
	END_IF
580:
	IF gICP.PDV.Get_Done_Ext() OR gICP.PDVOpenSensor THEN
		gRunningLog.append(CONCAT('Load Wafer POU Run:',DINT_TO_STRING(tempStep)));
		gRunningLog.append('Load Wafer POU Run:PDV Open Done');
		tempActStep.addStep(10,FALSE);
	END_IF
590:
	// 记忆状态更新
	gWaferMemoryState:=1;
	ups_CX51X0.Act_Wrtie();
	gRunningLog.append(CONCAT('Load Wafer POU Run:',DINT_TO_STRING(tempStep)));
	gRunningLog.append('Load Wafer POU Run:----Finish----');
	tempActStep.toDoneStep();
1000:
	tempActStep.toDoneStep();

60000://Done
	tempActStep.setDoneFlag();
	tempActStep.toZeroStep();
	
65000://Error
	tempActStep.setErrDoneFlag();
	tempActStep.toZeroStep();
	IF gICP.VentExtRelay THEN
		gICP.VentValve.Act_Retract();
	END_IF
END_CASE
END_METHOD

END_PROGRAM

// ---- POUs/MachinePOU/SemiAutomatic/S_RoughPumping.TcPOU
PROGRAM S_RoughPumping
VAR_INPUT
	bInit				:BOOL:=FALSE;// 初始化状态 busy/done/errDone
	bTrig				:BOOL:=FALSE;// 执行触发 信号
	bReset				:BOOL:=FALSE;// 报错 复位
	bPause				:BOOL:=FALSE;// 暂停 运行
	bStop				:BOOL:=FALSE;// 停止 运行
	bAbort				:BOOL:=FALSE;// 中止 运行
	
END_VAR
VAR_OUTPUT
	busy				:BOOL;
	done				:BOOL;
	errDone				:BOOL;
END_VAR
VAR
	actStep				:ActStepBase;
END_VAR
VAR
	i: INT;
	t1:ton;
	t2:ton;
	t3:ton;
	notchoose:BOOL;
	timeOutTime:TIME:=T#360S;
	safecheckTime:TIME:=T#1S;
END_VAR

busy:=actStep.isBusy();
done:=actStep.isDone();
errDone:=actStep.isError();
actStep.Act_Pause(pause:=bPause);

IF bTrig THEN
	bTrig:=FALSE;
	IF NOT busy THEN
		actStep.Act_ex();
	END_IF
END_IF

//状态复位
IF bInit THEN
	bInit:=FALSE;
	Act_init_status();
END_IF

IF bAbort OR bStop THEN
	bAbort:=FALSE;
	bStop:=FALSE;
	Act_init_status();
	actStep.toZeroStep();
	gShowLogTextTitle:='NON';
END_IF
ActionRun(tempActStep:=actStep);

(*
---Trigger action
*)
METHOD Act_Ex : BOOL
VAR_INPUT
END_VAR
IF NOT busy THEN
	actStep.Act_ex();
	Act_Ex:=TRUE;
ELSE
	Act_Ex:=FALSE;
END_IF
END_METHOD

(*
---功能: 状态复位 busy/done/errDone;
*)
METHOD Act_Init_Status
VAR_INPUT
END_VAR
actStep.Act_Init();
END_METHOD

METHOD PRIVATE ActionRun
VAR_INPUT
	tempActStep:ITFActStep;
END_VAR
VAR
END_VAR
VAR_STAT//此处定义静态变量, 保证每次进入该函数时能够在线监控当前值
	tempStep:DINT;
END_VAR
tempStep:=tempActStep.getStep();
CASE tempStep OF
0:
	IF tempActStep.isEx() THEN
		tempActStep.setBusyFlag();
		tempActStep.toBeginStep();
	END_IF
	t1(IN:= FALSE );
	t2(IN:= FALSE );
	t3(IN:= FALSE );
10:
	gShowLogTextTitle:='Rough Pumping';
	IF gRunningState<>RunningStatus.eErrorState THEN
		tempActStep.addStep(10,FALSE);
	ELSE
		error_Trigger(105);
		IF gCtrlMode=ControlMode.eManualCtrMode THEN
			tempActStep.toErrDoneStep();
		END_IF
	END_IF
20:
	IF NOT gICP.ForeLineGauge.error AND
		NOT gICP.LoadLockGauge.error  THEN
		tempActStep.addStep(80,FALSE);
	ELSE
		error_Trigger(107);
		IF gCtrlMode=ControlMode.eManualCtrMode THEN
			tempActStep.toErrDoneStep();
		END_IF
	END_IF
100:
	tempActStep.addStep(10,TRUE);
110:
	S_ActuatorRecoveryPOU.Act_Init_Status();
	S_ActuatorRecoveryPOU.Act_Ex();
	tempActStep.addStep(10,FALSE);
120:
	IF S_ActuatorRecoveryPOU.done THEN
		tempActStep.addStep(10,FALSE);
	END_IF
	IF S_ActuatorRecoveryPOU.errDone THEN
		tempActStep.toErrDoneStep();
	END_IF
130:
	tempActStep.addStep(10,FALSE);
140:
	gRunningLog.append('Rough Pumping POU Run:---Start---');
	IF NOT gRoughRemain THEN
		tempActStep.toStep(280,FALSE);
		gRunningLog.append(CONCAT('Rough Pumping POU Run:',DINT_TO_STRING(tempStep)));
		gRunningLog.append('Rough Pumping POU Run:RoughRemain has not been executed');
	ELSE
		tempActStep.toStep(510,FALSE);
		gRunningLog.append(CONCAT('Rough Pumping POU Run:',DINT_TO_STRING(tempStep)));
		gRunningLog.append('Rough Pumping POU Run:The -RoughRemain- has already been executed');
	END_IF
200:
	tempActStep.addStep(10,TRUE);
210:
	IF gICP.ForlinLineValve.Act_Extend() THEN
		gRunningLog.append(CONCAT('Rough Pumping POU Run:',DINT_TO_STRING(tempStep)));
		gRunningLog.append('Rough Pumping POU Run:FordLine Valve Open');
		tempActStep.addStep(10,FALSE);
	END_IF
220:
	IF gICP.ForlinLineValve.Get_Done_Ext() THEN
		gRunningLog.append(CONCAT('Rough Pumping POU Run:',DINT_TO_STRING(tempStep)));
		gRunningLog.append('Rough Pumping POU Run:ForeLine Valve Open Done');
		tempActStep.addStep(10,FALSE);
	END_IF
230:
	t2(IN:= gICP.ForeLineGauge.outputValue<gRoughtPumVaccum*10,PT:=safecheckTime*3 );
	IF t2.Q THEN
		t1(IN:= FALSE );
		t2(IN:= FALSE );
		t3(IN:= FALSE );
		gRunningLog.append(CONCAT('Rough Pumping POU Run:',DINT_TO_STRING(tempStep)));
		gRunningLog.append(CONCAT('Rough Pumping POU Run:ForeLine Pressure Arrive：',REAL_TO_STRING(gICP.ForeLineGauge.outputValue)));
		ups_CX51X0.Act_Wrtie();
		tempActStep.addStep(10,FALSE);
		RETURN;
	END_IF
	t1(IN:= TRUE,PT:=timeOutTime );
	IF t1.Q THEN
		t1(IN:= FALSE );
		t2(IN:= FALSE );
		t3(IN:= FALSE );
		error_Trigger(113);
		tempActStep.toStep(200,FALSE);
		RETURN;
	END_IF
240:
	tempActStep.addStep(10,TRUE);
250:
	IF gICP.ForlinLineValve.Act_Retract() THEN
		gRunningLog.append(CONCAT('Rough Pumping POU Run:',DINT_TO_STRING(tempStep)));
		gRunningLog.append('Rough Pumping POU Run:ForeLine Valve Close');
		tempActStep.addStep(10,FALSE);
	END_IF
260:
	IF gICP.ForlinLineValve.Get_Done_Ret() THEN
		gRunningLog.append(CONCAT('Rough Pumping POU Run:',DINT_TO_STRING(tempStep)));
		gRunningLog.append('Rough Pumping POU Run:ForeLine Valve Close Done');
		tempActStep.addStep(10,FALSE);
	END_IF
270:
	t3(IN:=TRUE,PT:=T#2S);
	IF t3.Q THEN
		t1(IN:= FALSE );
		t2(IN:= FALSE );
		t3(IN:= FALSE );
		tempActStep.toStep(360,FALSE);
	END_IF
280:
	tempActStep.addStep(10,TRUE);
290:
	IF gICP.RoughValve.Act_Extend() THEN
		gRunningLog.append(CONCAT('Rough Pumping POU Run:',DINT_TO_STRING(tempStep)));
		gRunningLog.append('Rough Pumping POU Run:Rough Valve Open');
		tempActStep.addStep(10,FALSE);
	END_IF
300:
	IF gICP.RoughValve.Get_Done_Ext() THEN
		gRunningLog.append(CONCAT('Rough Pumping POU Run:',DINT_TO_STRING(tempStep)));
		gRunningLog.append('Rough Pumping POU Run:Rough Valve Open Done');
		tempActStep.addStep(10,FALSE);
	END_IF
310:
	t2(IN:= gICP.ForeLineGauge.outputValue<gRoughtPumVaccum*10,PT:=safecheckTime*3 );
	IF t2.Q THEN
		t1(IN:= FALSE );
		t2(IN:= FALSE );
		t3(IN:= FALSE );
		gRunningLog.append(CONCAT('Rough Pumping POU Run:',DINT_TO_STRING(tempStep)));
		gRunningLog.append(CONCAT('Rough Pumping POU Run:Chamber Pressure Arrive：',REAL_TO_STRING(gICP.ForeLineGauge.outputValue)));
		tempActStep.addStep(10,FALSE);
		RETURN;
	END_IF
	t1(IN:= TRUE,PT:=timeOutTime );
	IF t1.Q THEN
		t1(IN:= FALSE );
		t2(IN:= FALSE );
		t3(IN:= FALSE );
		error_Trigger(113);
		tempActStep.toStep(280,FALSE);
		RETURN;
	END_IF
320:
	tempActStep.addStep(10,TRUE);
330:
	IF gICP.RoughValve.Act_Retract() THEN
		gRunningLog.append(CONCAT('Rough Pumping POU Run:',DINT_TO_STRING(tempStep)));
		gRunningLog.append('Rough Pumping POU Run:Rough Valve Close');
		tempActStep.addStep(10,FALSE);
	END_IF
340:
	IF gICP.RoughValve.Get_Done_Ret() THEN
		gRunningLog.append(CONCAT('Rough Pumping POU Run:',DINT_TO_STRING(tempStep)));
		gRunningLog.append('Rough Pumping POU Run:Rough Valve Close Done');
		tempActStep.addStep(10,FALSE);
	END_IF
350:
	t3(IN:=TRUE,PT:=T#2S);
	IF t3.Q THEN
		t1(IN:= FALSE );
		t2(IN:= FALSE );
		t3(IN:= FALSE );
		tempActStep.toStep(200,FALSE);
	END_IF
360:
	tempActStep.addStep(10,TRUE);
370:
	IF gICP.SlowPummingValve.Act_Extend() THEN
		gRunningLog.append(CONCAT('Rough Pumping POU Run:',DINT_TO_STRING(tempStep)));
		gRunningLog.append('Rough Pumping POU Run:SlowPump Valve Open');
		tempActStep.addStep(10,FALSE);
	END_IF
380:
	IF gICP.SlowPummingValve.Get_Done_Ext() THEN
		gRunningLog.append(CONCAT('Rough Pumping POU Run:',DINT_TO_STRING(tempStep)));
		gRunningLog.append('Rough Pumping POU Run:SlowPump Valve Open Done');
		tempActStep.addStep(10,FALSE);
	END_IF
390:
	t2(IN:= gICP.LoadLockGauge.outputValue<gLoadLockPumSVaccum,PT:=safecheckTime*3 );
	IF t2.Q THEN
		t1(IN:= FALSE );
		t2(IN:= FALSE );
		t3(IN:= FALSE );
		gRunningLog.append(CONCAT('Rough Pumping POU Run:',DINT_TO_STRING(tempStep)));
		gRunningLog.append(CONCAT('Rough Pumping POU Run:LoadLock Rough Pressure Arrive：',REAL_TO_STRING(gICP.LoadLockGauge.outputValue)));
		tempActStep.addStep(10,FALSE);
		RETURN;
	END_IF
	t1(IN:= TRUE,PT:=timeOutTime );
	IF t1.Q THEN
		t1(IN:= FALSE );
		t2(IN:= FALSE );
		t3(IN:= FALSE );
		error_Trigger(113);
		tempActStep.toStep(360,FALSE);
		RETURN;
	END_IF
400:
	tempActStep.addStep(10,TRUE);
410:
	IF gICP.SlowPummingValve.Act_Retract() THEN
		gRunningLog.append(CONCAT('Rough Pumping POU Run:',DINT_TO_STRING(tempStep)));
		gRunningLog.append('Rough Pumping POU Run:SlowPump Valve Close');
		tempActStep.addStep(10,FALSE);
	END_IF
420:
	IF gICP.SlowPummingValve.Get_Done_Ret() THEN
		gRunningLog.append(CONCAT('Rough Pumping POU Run:',DINT_TO_STRING(tempStep)));
		gRunningLog.append('Rough Pumping POU Run:SlowPump Valve Close Done');
		tempActStep.addStep(10,FALSE);
	END_IF
430:
	t3(IN:=TRUE,PT:=T#1S);
	IF t3.Q THEN
		t1(IN:= FALSE );
		t2(IN:= FALSE );
		t3(IN:= FALSE );
		tempActStep.addStep(10,FALSE);
	END_IF
440:
	tempActStep.addStep(10,TRUE);
450:
	IF gICP.FastPummingValve.Act_Extend() THEN
		gRunningLog.append(CONCAT('Rough Pumping POU Run:',DINT_TO_STRING(tempStep)));
		gRunningLog.append('Rough Pumping POU Run:FastwPump Valve Open');
		tempActStep.addStep(10,FALSE);
	END_IF
460:
	IF gICP.FastPummingValve.Get_Done_Ext() THEN
		gRunningLog.append(CONCAT('Rough Pumping POU Run:',DINT_TO_STRING(tempStep)));
		gRunningLog.append('Rough Pumping POU Run:FastwPump Valve Open Done');
		tempActStep.addStep(10,FALSE);
	END_IF
470:
	t2(IN:= gICP.LoadLockGauge.outputValue<gRoughtPumVaccum*2.5,PT:=safecheckTime );
	IF t2.Q THEN
		t1(IN:= FALSE );
		t2(IN:= FALSE );
		t3(IN:= FALSE );
		gRunningLog.append(CONCAT('Rough Pumping POU Run:',DINT_TO_STRING(tempStep)));
		gRunningLog.append(CONCAT('Rough Pumping POU Run:LoadLock Pressure Arrive：',REAL_TO_STRING(gICP.LoadLockGauge.outputValue)));
		
		tempActStep.addStep(10,FALSE);
		RETURN;
	END_IF
	t1(IN:= TRUE,PT:=timeOutTime );
	IF t1.Q THEN
		t1(IN:= FALSE );
		t2(IN:= FALSE );
		t3(IN:= FALSE );
		error_Trigger(113);
		tempActStep.toStep(440,FALSE);
		RETURN;
	END_IF
480:
	tempActStep.addStep(10,TRUE);
490:
	IF gICP.FastPummingValve.Act_Retract() THEN
		gRunningLog.append(CONCAT('Rough Pumping POU Run:',DINT_TO_STRING(tempStep)));
		gRunningLog.append('Rough Pumping POU Run:FastwPump Valve Close');
		tempActStep.addStep(10,FALSE);
	END_IF
500:
	IF gICP.FastPummingValve.Get_Done_Ret() THEN
		gRunningLog.append(CONCAT('Rough Pumping POU Run:',DINT_TO_STRING(tempStep)));
		gRunningLog.append('Rough Pumping POU Run:FastwPump Valve Close Done');
		tempActStep.addStep(10,FALSE);
	END_IF
510:
	t3(IN:=TRUE,PT:=T#2S);
	IF t3.Q THEN
		t1(IN:= FALSE );
		t2(IN:= FALSE );
		t3(IN:= FALSE );
		tempActStep.addStep(2,FALSE);
	END_IF
512:
	IF S_ActuatorRecoveryPOU.atmflag THEN
		S_BackOfHeliumClear.Act_Init_Status();
		S_BackOfHeliumClear.Act_Ex();
		tempActStep.addStep(2,FALSE);
	ELSE
		tempActStep.addStep(8,FALSE);
	END_IF
514:
	IF S_BackOfHeliumClear.busy THEN
		tempActStep.addStep(2,FALSE);
	END_IF
516:
	IF S_BackOfHeliumClear.done THEN
		tempActStep.addStep(2,FALSE);
	END_IF
518:
	tempActStep.addStep(2,FALSE);
520:
	IF gICP.ForlinLineValve.Act_Extend() AND gICP.PDV.Act_Open() THEN
		gRunningLog.append(CONCAT('Rough Pumping POU Run:',DINT_TO_STRING(tempStep)));
		gRunningLog.append('Rough Pumping POU Run:ForeLine Valve And PDV Open');
		tempActStep.addStep(10,FALSE);
	END_IF
530:
	IF gICP.ForlinLineValveExtRelay AND (gICP.PDV.Get_Done_Ext() OR gICP.PDVOpenSensor) THEN
		gRunningLog.append('Rough Pumping POU Run:ForLeine Valve And PDV Open Done');
		tempActStep.addStep(10,FALSE);
	END_IF
540:
	t3(IN:=TRUE,PT:=T#2S);
	IF t3.Q THEN
		t1(IN:= FALSE );
		t2(IN:= FALSE );
		t3(IN:= FALSE );
		tempActStep.addStep(10,FALSE);
	END_IF
550:
	tempActStep.toStep(1000,FALSE);
	IF NOT S_ChamberLLVent.busy AND NOT S_MachineVent.busy THEN
		gRoughRemain:=TRUE;
		gRoughRemainTMPCanOpen:=TRUE;
	END_IF
1000:
	tempActStep.toDoneStep();

60000://Done
	tempActStep.setDoneFlag();
	tempActStep.toZeroStep();
	S_ActuatorRecoveryPOU.atmflag:=FALSE;
	
65000://Error
	tempActStep.setErrDoneFlag();
	tempActStep.toZeroStep();
	S_ActuatorRecoveryPOU.atmflag:=FALSE;
END_CASE
END_METHOD

END_PROGRAM

// ---- POUs/MachinePOU/SemiAutomatic/S_BackOfHeliumClear.TcPOU
PROGRAM S_BackOfHeliumClear
VAR_INPUT
	bInit				:BOOL:=FALSE;// 初始化状态 busy/done/errDone
	bTrig				:BOOL:=FALSE;// 执行触发 信号
	bReset				:BOOL:=FALSE;// 报错 复位
	bPause				:BOOL:=FALSE;// 暂停 运行
	bStop				:BOOL:=FALSE;// 停止 运行
	bAbort				:BOOL:=FALSE;// 中止 运行
	
	atmflag:BOOL;
END_VAR
VAR_OUTPUT
	busy				:BOOL;
	done				:BOOL;
	errDone				:BOOL;
END_VAR
VAR
	actStep				:ActStepBase;
END_VAR
VAR
	i: INT;
	t1:ton;
	t2:ton;
	t3:ton;
	notchoose:BOOL;
//	str:STRING;
//	wstr:WSTRING;
END_VAR

busy:=actStep.isBusy();
done:=actStep.isDone();
errDone:=actStep.isError();
actStep.Act_Pause(pause:=bPause);

IF bTrig THEN
	bTrig:=FALSE;
	IF NOT busy THEN
		actStep.Act_ex();
	END_IF
END_IF

//状态复位
IF bInit THEN
	bInit:=FALSE;
	Act_init_status();
END_IF

IF bAbort OR bStop THEN
	bAbort:=FALSE;
	bStop:=FALSE;
	Act_init_status();
	actStep.toZeroStep();
	gShowLogTextTitle:='NON';
END_IF
ActionRun(tempActStep:=actStep);

(*
---Trigger action
*)
METHOD Act_Ex : BOOL
VAR_INPUT
END_VAR
IF NOT busy THEN
	actStep.Act_ex();
	Act_Ex:=TRUE;
ELSE
	Act_Ex:=FALSE;
END_IF
END_METHOD

(*
---功能: 状态复位 busy/done/errDone;
*)
METHOD Act_Init_Status
VAR_INPUT
END_VAR
actStep.Act_Init();
END_METHOD

METHOD PRIVATE ActionRun
VAR_INPUT
	tempActStep:ITFActStep;
END_VAR
VAR
END_VAR
VAR_STAT//此处定义静态变量, 保证每次进入该函数时能够在线监控当前值
	tempStep:DINT;
END_VAR
tempStep:=tempActStep.getStep();
CASE tempStep OF
0:
	IF tempActStep.isEx() THEN
		tempActStep.setBusyFlag();
		tempActStep.toBeginStep();
	END_IF
	t1(IN:= FALSE );
	t2(IN:= FALSE );
	t3(IN:= FALSE );
10:
	IF gICP.HeMFC_ActFlow<0.2 AND gICP.HeCheckGaugeReal<0.1 AND NOT gICP.HeINExtRelay AND NOT gICP.HePumExtRelay THEN
		tempActStep.toStep(430,FALSE);
		gRunningLog.append(CONCAT('He Actuator Recovery POU Run:',DINT_TO_STRING(tempStep)));
		gRunningLog.append('He Actuator Recovery POU Run: Back of helium clear done');
	ELSE
		tempActStep.addStep(10,FALSE);
		gRunningLog.append(CONCAT('He Actuator Recovery POU Run:',DINT_TO_STRING(tempStep)));
		gRunningLog.append('He Actuator Recovery POU Run: Back of helium not clear');
	END_IF
20:
	tempActStep.addStep(10,TRUE);
30:
	IF gICP.HeINValve.Act_Retract() THEN
		tempActStep.addStep(10,FALSE);
		gRunningLog.append(CONCAT('He Actuator Recovery POU Run:',DINT_TO_STRING(tempStep)));
		gRunningLog.append('He Actuator Recovery POU Run: HeIN Close');
	END_IF
40:
	IF gICP.HeINValve.Get_Done_Ret() THEN
		tempActStep.addStep(10,FALSE);
		gRunningLog.append(CONCAT('He Actuator Recovery POU Run:',DINT_TO_STRING(tempStep)));
		gRunningLog.append('He Actuator Recovery POU Run: HeIN Close');
	END_IF
50:
	tempActStep.addStep(10,TRUE);
60:
	IF gICP.HePumValve.Act_Extend() THEN
		tempActStep.addStep(10,FALSE);
		gRunningLog.append(CONCAT('He Actuator Recovery POU Run:',DINT_TO_STRING(tempStep)));
		gRunningLog.append('He Actuator Recovery POU Run: HePumValve Open');
	END_IF
70:
	IF gICP.HePumValve.Get_Done_Ext() THEN
		tempActStep.addStep(10,FALSE);
		gRunningLog.append(CONCAT('He Actuator Recovery POU Run:',DINT_TO_STRING(tempStep)));
		gRunningLog.append('He Actuator Recovery POU Run: HePumValve Open done');
	END_IF
80:
	t2(IN:=TRUE ,PT:=T#2S);
	IF t2.Q THEN
		t1(IN:= FALSE );
		t2(IN:= FALSE );
		t3(IN:= FALSE );
		tempActStep.addStep(10,FALSE);
	END_IF
90:
	t1(IN:=gICP.HeMFC_ActFlow<0.2 AND gICP.HeCheckGaugeReal<0.1 ,PT:=T#2S);
	IF t1.Q THEN
		t1(IN:= FALSE );
		t2(IN:= FALSE );
		t3(IN:= FALSE );
		gICP.HePumValve.Act_Retract();
		gRunningLog.append(CONCAT('He Actuator Recovery POU Run:',DINT_TO_STRING(tempStep)));
		gRunningLog.append('He Actuator Recovery POU Run: HePumValve close');
		tempActStep.addStep(10,FALSE);
	END_IF
100:
	IF gICP.HeINValve.Act_Retract() THEN
		tempActStep.addStep(10,FALSE);
		gRunningLog.append(CONCAT('He Actuator Recovery POU Run:',DINT_TO_STRING(tempStep)));
		gRunningLog.append('He Actuator Recovery POU Run: HePumValve close done');
	END_IF
110:
	IF gICP.HeINValve.Get_Done_Ret() THEN
		tempActStep.addStep(10,FALSE);
	END_IF
120:
	tempActStep.addStep(10,TRUE);
130:
	IF gICP.HePumValve.Act_Extend() THEN
		tempActStep.addStep(10,FALSE);
	END_IF
140:
	IF gICP.HePumValve.Get_Done_Ext() THEN
		tempActStep.addStep(10,FALSE);
	END_IF
150:
	t2(IN:=TRUE ,PT:=T#2S);
	IF t2.Q THEN
		t1(IN:= FALSE );
		t2(IN:= FALSE );
		t3(IN:= FALSE );
		tempActStep.addStep(10,FALSE);
	END_IF
160:
	t1(IN:=gICP.HeMFC_ActFlow<0.2AND gICP.HeCheckGaugeReal<0.1 AND gICP.ChamberGauge.outputValue1<500.0 AND NOT gICP.ChamberGauge.error,PT:=T#2S);
	IF t1.Q THEN
		t1(IN:= FALSE );
		t2(IN:= FALSE );
		t3(IN:= FALSE );
		gICP.HePumValve.Act_Retract();
		tempActStep.addStep(10,FALSE);
	END_IF
170:
	IF gICP.HePumValve.Get_Done_Ret() THEN
		tempActStep.addStep(10,FALSE);
	END_IF
180:
	tempActStep.toStep(430,FALSE);
430:
	tempActStep.toStep(1000,FALSE);
1000:
	tempActStep.toDoneStep();

60000://Done
	tempActStep.setDoneFlag();
	tempActStep.toZeroStep();
	
65000://Error
	tempActStep.setErrDoneFlag();
	tempActStep.toZeroStep();
	error_Trigger(300);
END_CASE
END_METHOD

END_PROGRAM

// ---- POUs/MachinePOU/SemiAutomatic/S_ChamberLLVent.TcPOU
PROGRAM S_ChamberLLVent
VAR_INPUT
	bInit				:BOOL:=FALSE;// 初始化状态 busy/done/errDone
	bTrig				:BOOL:=FALSE;// 执行触发 信号
	bReset				:BOOL:=FALSE;// 报错 复位
	bPause				:BOOL:=FALSE;// 暂停 运行
	bStop				:BOOL:=FALSE;// 停止 运行
	bAbort				:BOOL:=FALSE;// 中止 运行
	
END_VAR
VAR_OUTPUT
	busy				:BOOL;
	done				:BOOL;
	errDone				:BOOL;
END_VAR
VAR
	actStep				:ActStepBase;
END_VAR
VAR
	i: INT;
	t1:ton;
	t2:ton;
	t3:ton;
	notchoose:BOOL;
	timeOutTime:TIME:=T#120S;
	safecheckTime:TIME:=T#1S;
END_VAR

busy:=actStep.isBusy();
done:=actStep.isDone();
errDone:=actStep.isError();
actStep.Act_Pause(pause:=bPause);

IF bTrig THEN
	bTrig:=FALSE;
	IF NOT busy THEN
		actStep.Act_ex();
	END_IF
END_IF

//状态复位
IF bInit THEN
	bInit:=FALSE;
	Act_init_status();
END_IF

IF bAbort OR bStop THEN
	bAbort:=FALSE;
	bStop:=FALSE;
	Act_init_status();
	gShowLogTextTitle:='NON';
	actStep.toZeroStep();
END_IF
ActionRun(tempActStep:=actStep);

(*
---Trigger action
*)
METHOD Act_Ex : BOOL
VAR_INPUT
END_VAR
IF NOT busy THEN
	actStep.Act_ex();
	Act_Ex:=TRUE;
ELSE
	Act_Ex:=FALSE;
END_IF
END_METHOD

(*
---功能: 状态复位 busy/done/errDone;
*)
METHOD Act_Init_Status
VAR_INPUT
END_VAR
actStep.Act_Init();
END_METHOD

